LIN {X 0,Y 624.18,Z 1233.226,A -85,B 0,C 180,E1 28878.176,E2 28878.176} C_VEL
LIN {X 0,Y 624.369,Z 1226.316,A -85,B 0,C 180,E1 28876.192,E2 28876.192} C_VEL
LIN {X 0,Y 624.711,Z 1218.668,A -85,B 0,C 180,E1 28874.303,E2 28874.303} C_VEL
LIN {X 0,Y 625.236,Z 1208.486,A -85,B 0,C 180,E1 28872.115,E2 28872.115} C_VEL
LIN {X 0,Y 626.088,Z 1194.972,A -85,B 0,C 180,E1 28869.622,E2 28869.622} C_VEL
LIN {X 0,Y 627.007,Z 1182.374,A -85,B 0,C 180,E1 28867.593,E2 28867.593} C_VEL
LIN {X 0,Y 628.175,Z 1168.153,A -85,B 0,C 180,E1 28865.55,E2 28865.55} C_VEL
LIN {X 0,Y 629.836,Z 1149.568,A -85,B 0,C 180,E1 28863.198,E2 28863.198} C_VEL
LIN {X 0,Y 631.397,Z 1133.289,A -85,B 0,C 180,E1 28861.374,E2 28861.374} C_VEL
LIN {X 0,Y 633.134,Z 1116.14,A -85,B 0,C 180,E1 28859.642,E2 28859.642} C_VEL
LIN {X 0,Y 635.523,Z 1093.346,A -85,B 0,C 180,E1 28857.604,E2 28857.604} C_VEL
LIN {X 0,Y 637.441,Z 1075.082,A -85,B 0,C 180,E1 28856.159,E2 28856.159} C_VEL
LIN {X 0,Y 639.341,Z 1056.883,A -85,B 0,C 180,E1 28854.861,E2 28854.861} C_VEL
LIN {X 0,Y 641.452,Z 1036.313,A -85,B 0,C 180,E1 28853.547,E2 28853.547} C_VEL
LIN {X 0,Y 643.934,Z 1010.451,A -85,B 0,C 180,E1 28852.109,E2 28852.109} C_VEL
LIN {X 0,Y 645.904,Z 988.416,A -85,B 0,C 180,E1 28851.057,E2 28851.057} C_VEL
LIN {X 0,Y 647.711,Z 966.655,A -85,B 0,C 180,E1 28850.157,E2 28850.157} C_VEL
LIN {X 0,Y 649.668,Z 941.07,A -85,B 0,C 180,E1 28849.262,E2 28849.262} C_VEL
LIN {X 0,Y 651.274,Z 914.57,A -85,B 0,C 180,E1 28848.527,E2 28848.527} C_VEL
LIN {X 0,Y 652.424,Z 891.793,A -85,B 0,C 180,E1 28848.029,E2 28848.029} C_VEL
LIN {X 0,Y 653.308,Z 868.616,A -85,B 0,C 180,E1 28847.646,E2 28847.646} C_VEL
LIN {X 0,Y 657.558,Z 645.724,A -85,B 0,C 180,E1 28844.671,E2 28844.671} C_VEL
LIN {X 0,Y 661.46,Z 453.662,A -85,B 0,C 180,E1 28842.041,E2 28842.041} C_VEL
LIN {X 0,Y 652.442,Z 440.492,A -85,B 0,C 180,E1 28840.932,E2 28840.932} C_VEL
LIN {X 0,Y 640.565,Z 424.796,A -85,B 0,C 180,E1 28839.411,E2 28839.411} C_VEL
LIN {X 0,Y 636.522,Z 419.568,A -85,B 0,C 180,E1 28838.871,E2 28838.871} C_VEL
LIN {X 0,Y 632.798,Z 414.661,A -85,B 0,C 180,E1 28838.359,E2 28838.359} C_VEL
LIN {X 0,Y 629.914,Z 411.091,A -85,B 0,C 180,E1 28837.959,E2 28837.959} C_VEL
LIN {X 0,Y 628.864,Z 409.317,A -85,B 0,C 180,E1 28837.803,E2 28837.803} C_VEL
LIN {X 0,Y 626.22,Z 406.822,A -85,B 0,C 180,E1 28837.441,E2 28837.441} C_VEL
LIN {X 0,Y 624.999,Z 403.732,A -85,B 0,C 180,E1 28837.236,E2 28837.236} C_VEL
LIN {X 0,Y 624.947,Z 403.381,A -85,B 0,C 180,E1 28837.174,E2 28837.174} C_VEL
LIN {X 0,Y 624.942,Z 403.357,A -85,B 0,C 180,E1 28833.945,E2 28833.945} C_VEL
LIN {X 0,Y 624.938,Z 403.354,A -85,B 0,C 180,E1 28830.772,E2 28830.772} C_VEL
LIN {X 0,Y 624.939,Z 403.385,A -85,B 0,C 180,E1 28827.645,E2 28827.645} C_VEL
LIN {X 0,Y 624.94,Z 403.362,A -85,B 0,C 180,E1 28824.481,E2 28824.481} C_VEL
LIN {X 0,Y 624.932,Z 403.364,A -85,B 0,C 180,E1 28821.375,E2 28821.375} C_VEL
LIN {X 0,Y 624.944,Z 403.382,A -85,B 0,C 180,E1 28818.276,E2 28818.276} C_VEL
LIN {X 0,Y 624.926,Z 403.352,A -85,B 0,C 180,E1 28815.118,E2 28815.118} C_VEL
LIN {X 0,Y 624.945,Z 403.387,A -85,B 0,C 180,E1 28812.005,E2 28812.005} C_VEL
LIN {X 0,Y 624.923,Z 403.347,A -85,B 0,C 180,E1 28808.836,E2 28808.836} C_VEL
LIN {X 0,Y 624.946,Z 403.385,A -85,B 0,C 180,E1 28805.785,E2 28805.785} C_VEL
LIN {X 0,Y 624.921,Z 403.345,A -85,B 0,C 180,E1 28802.66,E2 28802.66} C_VEL
LIN {X 0,Y 624.949,Z 403.386,A -85,B 0,C 180,E1 28799.633,E2 28799.633} C_VEL
LIN {X 0,Y 624.922,Z 403.343,A -85,B 0,C 180,E1 28796.514,E2 28796.514} C_VEL
LIN {X 0,Y 624.948,Z 403.382,A -85,B 0,C 180,E1 28793.385,E2 28793.385} C_VEL
LIN {X 0,Y 624.918,Z 403.35,A -85,B 0,C 180,E1 28790.235,E2 28790.235} C_VEL
LIN {X 0,Y 624.949,Z 403.377,A -85,B 0,C 180,E1 28787.15,E2 28787.15} C_VEL
LIN {X 0,Y 624.919,Z 403.366,A -85,B 0,C 180,E1 28784.026,E2 28784.026} C_VEL
LIN {X 0,Y 624.948,Z 403.363,A -85,B 0,C 180,E1 28780.95,E2 28780.95} C_VEL
LIN {X 0,Y 624.918,Z 403.383,A -85,B 0,C 180,E1 28777.814,E2 28777.814} C_VEL
LIN {X 0,Y 624.947,Z 403.352,A -85,B 0,C 180,E1 28774.711,E2 28774.711} C_VEL
LIN {X 0,Y 624.917,Z 403.38,A -85,B 0,C 180,E1 28771.627,E2 28771.627} C_VEL
LIN {X 0,Y 624.954,Z 403.379,A -85,B 0,C 180,E1 28768.561,E2 28768.561} C_VEL
LIN {X 0,Y 624.916,Z 403.363,A -85,B 0,C 180,E1 28765.388,E2 28765.388} C_VEL
LIN {X 0,Y 624.957,Z 403.626,A -85,B 0,C 180,E1 28764.832,E2 28764.832} C_VEL
LIN {X 0,Y 626.263,Z 406.877,A -85,B 0,C 180,E1 28764.355,E2 28764.355} C_VEL
LIN {X 0,Y 627.353,Z 408.515,A -85,B 0,C 180,E1 28764.065,E2 28764.065} C_VEL
LIN {X 0,Y 629.05,Z 412.084,A -85,B 0,C 180,E1 28763.524,E2 28763.524} C_VEL
LIN {X 0,Y 634.263,Z 422.738,A -85,B 0,C 180,E1 28761.946,E2 28761.946} C_VEL
LIN {X 0,Y 636.116,Z 426.172,A -85,B 0,C 180,E1 28761.475,E2 28761.475} C_VEL
LIN {X 0,Y 652.475,Z 449.581,A -85,B 0,C 180,E1 28759.332,E2 28759.332} C_VEL
LIN {X 0,Y 661.483,Z 463.146,A -85,B 0,C 180,E1 28758.223,E2 28758.223} C_VEL
LIN {X 0,Y 661.775,Z 465.886,A -85,B 0,C 180,E1 28758.151,E2 28758.151} C_VEL
LIN {X 0,Y 657.599,Z 673.657,A -85,B 0,C 180,E1 28755.311,E2 28755.311} C_VEL
LIN {X 0,Y 653.346,Z 897.515,A -85,B 0,C 180,E1 28752.325,E2 28752.325} C_VEL
LIN {X 0,Y 652.452,Z 921.239,A -85,B 0,C 180,E1 28751.936,E2 28751.936} C_VEL
LIN {X 0,Y 651.313,Z 943.825,A -85,B 0,C 180,E1 28751.446,E2 28751.446} C_VEL
LIN {X 0,Y 649.785,Z 969.298,A -85,B 0,C 180,E1 28750.747,E2 28750.747} C_VEL
LIN {X 0,Y 647.795,Z 995.651,A -85,B 0,C 180,E1 28749.836,E2 28749.836} C_VEL
LIN {X 0,Y 645.982,Z 1017.523,A -85,B 0,C 180,E1 28748.937,E2 28748.937} C_VEL
LIN {X 0,Y 644.092,Z 1038.646,A -85,B 0,C 180,E1 28747.936,E2 28747.936} C_VEL
LIN {X 0,Y 641.751,Z 1063.464,A -85,B 0,C 180,E1 28746.584,E2 28746.584} C_VEL
LIN {X 0,Y 639.401,Z 1086.279,A -85,B 0,C 180,E1 28745.136,E2 28745.136} C_VEL
LIN {X 0,Y 637.5,Z 1104.526,A -85,B 0,C 180,E1 28743.838,E2 28743.838} C_VEL
LIN {X 0,Y 635.638,Z 1122.229,A -85,B 0,C 180,E1 28742.442,E2 28742.442} C_VEL
LIN {X 0,Y 633.467,Z 1143.165,A -85,B 0,C 180,E1 28740.603,E2 28740.603} C_VEL
LIN {X 0,Y 631.479,Z 1162.423,A -85,B 0,C 180,E1 28738.673,E2 28738.673} C_VEL
LIN {X 0,Y 629.929,Z 1178.632,A -85,B 0,C 180,E1 28736.865,E2 28736.865} C_VEL
LIN {X 0,Y 628.322,Z 1196.412,A -85,B 0,C 180,E1 28734.644,E2 28734.644} C_VEL
LIN {X 0,Y 627.081,Z 1211.45,A -85,B 0,C 180,E1 28732.503,E2 28732.503} C_VEL
LIN {X 0,Y 626.139,Z 1224.134,A -85,B 0,C 180,E1 28730.474,E2 28730.474} C_VEL
LIN {X 0,Y 625.299,Z 1237.338,A -85,B 0,C 180,E1 28728.076,E2 28728.076} C_VEL
LIN {X 0,Y 624.747,Z 1248.064,A -85,B 0,C 180,E1 28725.791,E2 28725.791} C_VEL
LIN {X 0,Y 624.373,Z 1256.146,A -85,B 0,C 180,E1 28723.808,E2 28723.808} C_VEL
LIN {X 0,Y 624.185,Z 1262.738,A -85,B 0,C 180,E1 28721.929,E2 28721.929} C_VEL
LIN {X 0,Y 624.025,Z 1268.81,A -85,B 0,C 180,E1 28719.876,E2 28719.876} C_VEL
LIN {X 0,Y 623.936,Z 1274.143,A -85,B 0,C 180,E1 28717.647,E2 28717.647} C_VEL
LIN {X 0,Y 623.92,Z 1278.422,A -85,B 0,C 180,E1 28715.153,E2 28715.153} C_VEL
LIN {X 0,Y 623.91,Z 1280.741,A -85,B 0,C 180,E1 28712.944,E2 28712.944} C_VEL
LIN {X 0,Y 623.875,Z 1281.759,A -85,B 0,C 180,E1 28711.014,E2 28711.014} C_VEL
LIN {X 0,Y 623.865,Z 1281.806,A -85,B 0,C 180,E1 28709.178,E2 28709.178} C_VEL
LIN {X 0,Y 623.909,Z 1280.95,A -85,B 0,C 180,E1 28707.341,E2 28707.341} C_VEL
LIN {X 0,Y 623.915,Z 1278.904,A -85,B 0,C 180,E1 28705.224,E2 28705.224} C_VEL
LIN {X 0,Y 623.953,Z 1275.087,A -85,B 0,C 180,E1 28702.824,E2 28702.824} C_VEL
LIN {X 0,Y 623.985,Z 1269.85,A -85,B 0,C 180,E1 28700.505,E2 28700.505} C_VEL
LIN {X 0,Y 624.178,Z 1263.371,A -85,B 0,C 180,E1 28698.266,E2 28698.266} C_VEL
LIN {X 0,Y 624.361,Z 1256.533,A -85,B 0,C 180,E1 28696.295,E2 28696.295} C_VEL
LIN {X 0,Y 624.7,Z 1248.923,A -85,B 0,C 180,E1 28694.407,E2 28694.407} C_VEL
LIN {X 0,Y 625.201,Z 1239.245,A -85,B 0,C 180,E1 28692.315,E2 28692.315} C_VEL
LIN {X 0,Y 626.033,Z 1225.91,A -85,B 0,C 180,E1 28689.824,E2 28689.824} C_VEL
LIN {X 0,Y 627.001,Z 1212.516,A -85,B 0,C 180,E1 28687.66,E2 28687.66} C_VEL
LIN {X 0,Y 628.135,Z 1198.609,A -85,B 0,C 180,E1 28685.658,E2 28685.658} C_VEL
LIN {X 0,Y 629.782,Z 1180.116,A -85,B 0,C 180,E1 28683.307,E2 28683.307} C_VEL
LIN {X 0,Y 631.386,Z 1163.434,A -85,B 0,C 180,E1 28681.435,E2 28681.435} C_VEL
LIN {X 0,Y 633.123,Z 1146.245,A -85,B 0,C 180,E1 28679.697,E2 28679.697} C_VEL
LIN {X 0,Y 635.505,Z 1123.499,A -85,B 0,C 180,E1 28677.662,E2 28677.662} C_VEL
LIN {X 0,Y 637.379,Z 1105.658,A -85,B 0,C 180,E1 28676.247,E2 28676.247} C_VEL
LIN {X 0,Y 639.312,Z 1087.141,A -85,B 0,C 180,E1 28674.924,E2 28674.924} C_VEL
LIN {X 0,Y 641.394,Z 1066.854,A -85,B 0,C 180,E1 28673.625,E2 28673.625} C_VEL
LIN {X 0,Y 643.903,Z 1040.838,A -85,B 0,C 180,E1 28672.174,E2 28672.174} C_VEL
LIN {X 0,Y 645.857,Z 1018.977,A -85,B 0,C 180,E1 28671.127,E2 28671.127} C_VEL
LIN {X 0,Y 647.601,Z 998.036,A -85,B 0,C 180,E1 28670.256,E2 28670.256} C_VEL
LIN {X 0,Y 649.259,Z 976.12,A -85,B 0,C 180,E1 28669.474,E2 28669.474} C_VEL
LIN {X 0,Y 651.057,Z 948.853,A -85,B 0,C 180,E1 28668.675,E2 28668.675} C_VEL
LIN {X 0,Y 652.353,Z 923.503,A -85,B 0,C 180,E1 28668.107,E2 28668.107} C_VEL
LIN {X 0,Y 653.236,Z 900.82,A -85,B 0,C 180,E1 28667.723,E2 28667.723} C_VEL
LIN {X 0,Y 657.425,Z 682.671,A -85,B 0,C 180,E1 28664.81,E2 28664.81} C_VEL
LIN {X 0,Y 661.622,Z 473.319,A -85,B 0,C 180,E1 28661.952,E2 28661.952} C_VEL
LIN {X 0,Y 661.642,Z 463.826,A -85,B 0,C 180,E1 28661.803,E2 28661.803} C_VEL
LIN {X 0,Y 660.917,Z 462.029,A -85,B 0,C 180,E1 28661.705,E2 28661.705} C_VEL
LIN {X 0,Y 647.235,Z 442.165,A -85,B 0,C 180,E1 28660.005,E2 28660.005} C_VEL
LIN {X 0,Y 635.569,Z 425.222,A -85,B 0,C 180,E1 28658.42,E2 28658.42} C_VEL
LIN {X 0,Y 630.828,Z 415.845,A -85,B 0,C 180,E1 28657.036,E2 28657.036} C_VEL
LIN {X 0,Y 628.688,Z 411.575,A -85,B 0,C 180,E1 28656.387,E2 28656.387} C_VEL
LIN {X 0,Y 626.981,Z 407.792,A -85,B 0,C 180,E1 28655.823,E2 28655.823} C_VEL
LIN {X 0,Y 625.107,Z 404.452,A -85,B 0,C 180,E1 28655.271,E2 28655.271} C_VEL
LIN {X 0,Y 624.89,Z 403.378,A -85,B 0,C 180,E1 28655.101,E2 28655.101} C_VEL
LIN {X 0,Y 624.932,Z 403.383,A -85,B 0,C 180,E1 28652.191,E2 28652.191} C_VEL
LIN {X 0,Y 624.885,Z 403.365,A -85,B 0,C 180,E1 28649.107,E2 28649.107} C_VEL
LIN {X 0,Y 624.886,Z 403.376,A -85,B 0,C 180,E1 28646.413,E2 28646.413} C_VEL
LIN {X 0,Y 624.898,Z 403.391,A -85,B 0,C 180,E1 28643.18,E2 28643.18} C_VEL
LIN {X 0,Y 624.865,Z 403.359,A -85,B 0,C 180,E1 28640.514,E2 28640.514} C_VEL
LIN {X 0,Y 624.944,Z 403.389,A -85,B 0,C 180,E1 28637.505,E2 28637.505} C_VEL
LIN {X 0,Y 624.855,Z 403.36,A -85,B 0,C 180,E1 28634.537,E2 28634.537} C_VEL
LIN {X 0,Y 624.882,Z 403.392,A -85,B 0,C 180,E1 28631.819,E2 28631.819} C_VEL
LIN {X 0,Y 624.852,Z 403.363,A -85,B 0,C 180,E1 28628.586,E2 28628.586} C_VEL
LIN {X 0,Y 624.848,Z 403.394,A -85,B 0,C 180,E1 28626.063,E2 28626.063} C_VEL
LIN {X 0,Y 624.921,Z 403.351,A -85,B 0,C 180,E1 28623.027,E2 28623.027} C_VEL
LIN {X 0,Y 624.858,Z 403.393,A -85,B 0,C 180,E1 28620.092,E2 28620.092} C_VEL
LIN {X 0,Y 624.91,Z 403.353,A -85,B 0,C 180,E1 28617.249,E2 28617.249} C_VEL
LIN {X 0,Y 624.872,Z 403.391,A -85,B 0,C 180,E1 28614.122,E2 28614.122} C_VEL
LIN {X 0,Y 624.883,Z 403.359,A -85,B 0,C 180,E1 28611.442,E2 28611.442} C_VEL
LIN {X 0,Y 624.896,Z 403.389,A -85,B 0,C 180,E1 28608.181,E2 28608.181} C_VEL
LIN {X 0,Y 624.883,Z 403.358,A -85,B 0,C 180,E1 28605.45,E2 28605.45} C_VEL
LIN {X 0,Y 624.936,Z 403.386,A -85,B 0,C 180,E1 28602.302,E2 28602.302} C_VEL
LIN {X 0,Y 624.888,Z 403.354,A -85,B 0,C 180,E1 28599.38,E2 28599.38} C_VEL
LIN {X 0,Y 624.954,Z 403.378,A -85,B 0,C 180,E1 28596.323,E2 28596.323} C_VEL
LIN {X 0,Y 624.898,Z 403.371,A -85,B 0,C 180,E1 28593.28,E2 28593.28} C_VEL
LIN {X 0,Y 624.953,Z 403.353,A -85,B 0,C 180,E1 28590.265,E2 28590.265} C_VEL
LIN {X 0,Y 624.908,Z 403.391,A -85,B 0,C 180,E1 28587.151,E2 28587.151} C_VEL
LIN {X 0,Y 624.951,Z 403.371,A -85,B 0,C 180,E1 28584.042,E2 28584.042} C_VEL
LIN {X 0,Y 624.961,Z 403.612,A -85,B 0,C 180,E1 28582.679,E2 28582.679} C_VEL
LIN {X 0,Y 626.132,Z 406.672,A -85,B 0,C 180,E1 28582.48,E2 28582.48} C_VEL
LIN {X 0,Y 628.699,Z 409.185,A -85,B 0,C 180,E1 28582.128,E2 28582.128} C_VEL
LIN {X 0,Y 629.507,Z 410.299,A -85,B 0,C 180,E1 28582.012,E2 28582.012} C_VEL
LIN {X 0,Y 632.071,Z 413.977,A -85,B 0,C 180,E1 28581.646,E2 28581.646} C_VEL
LIN {X 0,Y 633.818,Z 415.911,A -85,B 0,C 180,E1 28581.411,E2 28581.411} C_VEL
LIN {X 0,Y 637.218,Z 420.26,A -85,B 0,C 180,E1 28580.949,E2 28580.949} C_VEL
LIN {X 0,Y 651.261,Z 439.003,A -85,B 0,C 180,E1 28579.123,E2 28579.123} C_VEL
LIN {X 0,Y 660.214,Z 451.648,A -85,B 0,C 180,E1 28578.022,E2 28578.022} C_VEL
LIN {X 0,Y 661.481,Z 454.083,A -85,B 0,C 180,E1 28577.86,E2 28577.86} C_VEL
LIN {X 0,Y 660.474,Z 501.439,A -85,B 0,C 180,E1 28577.206,E2 28577.206} C_VEL
LIN {X 0,Y 659.621,Z 509.147,A -85,B 0,C 180,E1 28577.165,E2 28577.165} C_VEL
LIN {X 0,Y 654.944,Z 529.83,A -85,B 0,C 180,E1 28577.283,E2 28577.283} C_VEL
LIN {X 0,Y 654.301,Z 536.437,A -85,B 0,C 180,E1 28577.239,E2 28577.239} C_VEL
LIN {X 0,Y 649.641,Z 757.843,A -85,B 0,C 180,E1 28574.227,E2 28574.227} C_VEL
LIN {X 0,Y 647.176,Z 874.928,A -85,B 0,C 180,E1 28572.649,E2 28572.649} C_VEL
LIN {X 0,Y 646,Z 902.071,A -85,B 0,C 180,E1 28572.153,E2 28572.153} C_VEL
LIN {X 0,Y 644.375,Z 928.231,A -85,B 0,C 180,E1 28571.496,E2 28571.496} C_VEL
LIN {X 0,Y 642.849,Z 949.425,A -85,B 0,C 180,E1 28570.839,E2 28570.839} C_VEL
LIN {X 0,Y 641.18,Z 970.031,A -85,B 0,C 180,E1 28570.087,E2 28570.087} C_VEL
LIN {X 0,Y 639.218,Z 992.171,A -85,B 0,C 180,E1 28569.145,E2 28569.145} C_VEL
LIN {X 0,Y 636.642,Z 1018.743,A -85,B 0,C 180,E1 28567.814,E2 28567.814} C_VEL
LIN {X 0,Y 634.448,Z 1039.446,A -85,B 0,C 180,E1 28566.613,E2 28566.613} C_VEL
LIN {X 0,Y 632.414,Z 1058.012,A -85,B 0,C 180,E1 28565.405,E2 28565.405} C_VEL
LIN {X 0,Y 630.33,Z 1076.763,A -85,B 0,C 180,E1 28564.046,E2 28564.046} C_VEL
LIN {X 0,Y 627.864,Z 1098.737,A -85,B 0,C 180,E1 28562.26,E2 28562.26} C_VEL
LIN {X 0,Y 625.641,Z 1118.412,A -85,B 0,C 180,E1 28560.432,E2 28560.432} C_VEL
LIN {X 0,Y 623.881,Z 1134.672,A -85,B 0,C 180,E1 28558.756,E2 28558.756} C_VEL
LIN {X 0,Y 621.996,Z 1153.107,A -85,B 0,C 180,E1 28556.641,E2 28556.641} C_VEL
LIN {X 0,Y 620.362,Z 1170.144,A -85,B 0,C 180,E1 28554.403,E2 28554.403} C_VEL
LIN {X 0,Y 619.177,Z 1183.762,A -85,B 0,C 180,E1 28552.396,E2 28552.396} C_VEL
LIN {X 0,Y 618.058,Z 1198.42,A -85,B 0,C 180,E1 28549.954,E2 28549.954} C_VEL
LIN {X 0,Y 617.254,Z 1210.428,A -85,B 0,C 180,E1 28547.628,E2 28547.628} C_VEL
LIN {X 0,Y 616.73,Z 1219.949,A -85,B 0,C 180,E1 28545.511,E2 28545.511} C_VEL
LIN {X 0,Y 616.358,Z 1228.838,A -85,B 0,C 180,E1 28543.218,E2 28543.218} C_VEL
LIN {X 0,Y 616.104,Z 1236.923,A -85,B 0,C 180,E1 28540.657,E2 28540.657} C_VEL
LIN {X 0,Y 615.995,Z 1242.642,A -85,B 0,C 180,E1 28538.396,E2 28538.396} C_VEL
LIN {X 0,Y 615.936,Z 1247.124,A -85,B 0,C 180,E1 28536.052,E2 28536.052} C_VEL
LIN {X 0,Y 615.913,Z 1250.306,A -85,B 0,C 180,E1 28533.532,E2 28533.532} C_VEL
LIN {X 0,Y 615.894,Z 1251.704,A -85,B 0,C 180,E1 28531.205,E2 28531.205} C_VEL
LIN {X 0,Y 615.864,Z 1251.837,A -85,B 0,C 180,E1 28529.252,E2 28529.252} C_VEL
LIN {X 0,Y 615.907,Z 1250.977,A -85,B 0,C 180,E1 28527.297,E2 28527.297} C_VEL
LIN {X 0,Y 615.915,Z 1248.946,A -85,B 0,C 180,E1 28525.153,E2 28525.153} C_VEL
LIN {X 0,Y 615.954,Z 1245.154,A -85,B 0,C 180,E1 28522.722,E2 28522.722} C_VEL
LIN {X 0,Y 616.007,Z 1239.693,A -85,B 0,C 180,E1 28520.278,E2 28520.278} C_VEL
LIN {X 0,Y 616.197,Z 1233.451,A -85,B 0,C 180,E1 28518.092,E2 28518.092} C_VEL
LIN {X 0,Y 616.402,Z 1226.667,A -85,B 0,C 180,E1 28516.105,E2 28516.105} C_VEL
LIN {X 0,Y 616.772,Z 1219.075,A -85,B 0,C 180,E1 28514.192,E2 28514.192} C_VEL
LIN {X 0,Y 617.303,Z 1209.416,A -85,B 0,C 180,E1 28512.073,E2 28512.073} C_VEL
LIN {X 0,Y 618.211,Z 1196.113,A -85,B 0,C 180,E1 28509.549,E2 28509.549} C_VEL
LIN {X 0,Y 619.232,Z 1183.003,A -85,B 0,C 180,E1 28507.396,E2 28507.396} C_VEL
LIN {X 0,Y 620.417,Z 1169.572,A -85,B 0,C 180,E1 28505.427,E2 28505.427} C_VEL
LIN {X 0,Y 622.116,Z 1151.935,A -85,B 0,C 180,E1 28503.129,E2 28503.129} C_VEL
LIN {X 0,Y 623.88,Z 1134.67,A -85,B 0,C 180,E1 28501.154,E2 28501.154} C_VEL
LIN {X 0,Y 625.64,Z 1118.409,A -85,B 0,C 180,E1 28499.477,E2 28499.477} C_VEL
LIN {X 0,Y 627.941,Z 1098.152,A -85,B 0,C 180,E1 28497.598,E2 28497.598} C_VEL
LIN {X 0,Y 630.37,Z 1076.407,A -85,B 0,C 180,E1 28495.837,E2 28495.837} C_VEL
LIN {X 0,Y 632.454,Z 1057.679,A -85,B 0,C 180,E1 28494.482,E2 28494.482} C_VEL
LIN {X 0,Y 634.5,Z 1038.978,A -85,B 0,C 180,E1 28493.268,E2 28493.268} C_VEL
LIN {X 0,Y 637.003,Z 1015.386,A -85,B 0,C 180,E1 28491.909,E2 28491.909} C_VEL
LIN {X 0,Y 639.342,Z 990.659,A -85,B 0,C 180,E1 28490.697,E2 28490.697} C_VEL
LIN {X 0,Y 641.244,Z 969.205,A -85,B 0,C 180,E1 28489.791,E2 28489.791} C_VEL
LIN {X 0,Y 642.921,Z 948.454,A -85,B 0,C 180,E1 28489.038,E2 28489.038} C_VEL
LIN {X 0,Y 644.672,Z 924.03,A -85,B 0,C 180,E1 28488.293,E2 28488.293} C_VEL
LIN {X 0,Y 646.263,Z 895.924,A -85,B 0,C 180,E1 28487.633,E2 28487.633} C_VEL
LIN {X 0,Y 647.247,Z 872.707,A -85,B 0,C 180,E1 28487.228,E2 28487.228} C_VEL
LIN {X 0,Y 651.601,Z 661.791,A -85,B 0,C 180,E1 28484.388,E2 28484.388} C_VEL
LIN {X 0,Y 656.051,Z 457.437,A -85,B 0,C 180,E1 28481.572,E2 28481.572} C_VEL
LIN {X 0,Y 645.173,Z 442.024,A -85,B 0,C 180,E1 28480.203,E2 28480.203} C_VEL
LIN {X 0,Y 633.088,Z 426.146,A -85,B 0,C 180,E1 28478.599,E2 28478.599} C_VEL
LIN {X 0,Y 629.106,Z 421.023,A -85,B 0,C 180,E1 28478.045,E2 28478.045} C_VEL
LIN {X 0,Y 625.872,Z 416.621,A -85,B 0,C 180,E1 28477.581,E2 28477.581} C_VEL
LIN {X 0,Y 622.34,Z 412.611,A -85,B 0,C 180,E1 28477.078,E2 28477.078} C_VEL
LIN {X 0,Y 621.204,Z 410.46,A -85,B 0,C 180,E1 28476.897,E2 28476.897} C_VEL
LIN {X 0,Y 618.464,Z 408.085,A -85,B 0,C 180,E1 28476.51,E2 28476.51} C_VEL
LIN {X 0,Y 617.116,Z 405.016,A -85,B 0,C 180,E1 28476.28,E2 28476.28} C_VEL
LIN {X 0,Y 617.01,Z 404.371,A -85,B 0,C 180,E1 28476.227,E2 28476.227} C_VEL
LIN {X 0,Y 617.009,Z 404.366,A -85,B 0,C 180,E1 28472.991,E2 28472.991} C_VEL
LIN {X 0,Y 616.998,Z 404.342,A -85,B 0,C 180,E1 28469.729,E2 28469.729} C_VEL
LIN {X 0,Y 617.004,Z 404.351,A -85,B 0,C 180,E1 28466.673,E2 28466.673} C_VEL
LIN {X 0,Y 616.996,Z 404.37,A -85,B 0,C 180,E1 28463.47,E2 28463.47} C_VEL
LIN {X 0,Y 617.004,Z 404.337,A -85,B 0,C 180,E1 28460.391,E2 28460.391} C_VEL
LIN {X 0,Y 616.995,Z 404.373,A -85,B 0,C 180,E1 28457.252,E2 28457.252} C_VEL
LIN {X 0,Y 617.005,Z 404.339,A -85,B 0,C 180,E1 28454.164,E2 28454.164} C_VEL
LIN {X 0,Y 616.993,Z 404.372,A -85,B 0,C 180,E1 28451.025,E2 28451.025} C_VEL
LIN {X 0,Y 617.002,Z 404.343,A -85,B 0,C 180,E1 28447.824,E2 28447.824} C_VEL
LIN {X 0,Y 616.986,Z 404.369,A -85,B 0,C 180,E1 28444.666,E2 28444.666} C_VEL
LIN {X 0,Y 617.003,Z 404.348,A -85,B 0,C 180,E1 28441.486,E2 28441.486} C_VEL
LIN {X 0,Y 616.983,Z 404.365,A -85,B 0,C 180,E1 28438.421,E2 28438.421} C_VEL
LIN {X 0,Y 617.003,Z 404.35,A -85,B 0,C 180,E1 28435.259,E2 28435.259} C_VEL
LIN {X 0,Y 616.98,Z 404.359,A -85,B 0,C 180,E1 28432.176,E2 28432.176} C_VEL
LIN {X 0,Y 617.007,Z 404.357,A -85,B 0,C 180,E1 28429.07,E2 28429.07} C_VEL
LIN {X 0,Y 616.977,Z 404.349,A -85,B 0,C 180,E1 28425.931,E2 28425.931} C_VEL
LIN {X 0,Y 617.01,Z 404.373,A -85,B 0,C 180,E1 28422.846,E2 28422.846} C_VEL
LIN {X 0,Y 616.975,Z 404.34,A -85,B 0,C 180,E1 28419.707,E2 28419.707} C_VEL
LIN {X 0,Y 617.01,Z 404.367,A -85,B 0,C 180,E1 28416.607,E2 28416.607} C_VEL
LIN {X 0,Y 616.975,Z 404.363,A -85,B 0,C 180,E1 28413.43,E2 28413.43} C_VEL
LIN {X 0,Y 617.01,Z 404.339,A -85,B 0,C 180,E1 28410.379,E2 28410.379} C_VEL
LIN {X 0,Y 616.972,Z 404.36,A -85,B 0,C 180,E1 28407.26,E2 28407.26} C_VEL
LIN {X 0,Y 617.022,Z 404.501,A -85,B 0,C 180,E1 28405.758,E2 28405.758} C_VEL
LIN {X 0,Y 618.161,Z 407.659,A -85,B 0,C 180,E1 28405.294,E2 28405.294} C_VEL
LIN {X 0,Y 619.485,Z 409.717,A -85,B 0,C 180,E1 28404.921,E2 28404.921} C_VEL
LIN {X 0,Y 626.365,Z 423.493,A -85,B 0,C 180,E1 28402.77,E2 28402.77} C_VEL
LIN {X 0,Y 627.636,Z 425.839,A -85,B 0,C 180,E1 28402.456,E2 28402.456} C_VEL
LIN {X 0,Y 639.368,Z 442.419,A -85,B 0,C 180,E1 28400.831,E2 28400.831} C_VEL
LIN {X 0,Y 652.071,Z 460.969,A -85,B 0,C 180,E1 28399.185,E2 28399.185} C_VEL
LIN {X 0,Y 656.372,Z 467.664,A -85,B 0,C 180,E1 28398.648,E2 28398.648} C_VEL
LIN {X 0,Y 651.927,Z 675.488,A -85,B 0,C 180,E1 28395.788,E2 28395.788} C_VEL
LIN {X 0,Y 647.408,Z 898.124,A -85,B 0,C 180,E1 28392.795,E2 28392.795} C_VEL
LIN {X 0,Y 646.478,Z 921.376,A -85,B 0,C 180,E1 28392.41,E2 28392.41} C_VEL
LIN {X 0,Y 645.285,Z 943.689,A -85,B 0,C 180,E1 28391.924,E2 28391.924} C_VEL
LIN {X 0,Y 643.695,Z 968.754,A -85,B 0,C 180,E1 28391.235,E2 28391.235} C_VEL
LIN {X 0,Y 641.555,Z 995.648,A -85,B 0,C 180,E1 28390.303,E2 28390.303} C_VEL
LIN {X 0,Y 639.631,Z 1017.52,A -85,B 0,C 180,E1 28389.398,E2 28389.398} C_VEL
LIN {X 0,Y 637.621,Z 1038.642,A -85,B 0,C 180,E1 28388.391,E2 28388.391} C_VEL
LIN {X 0,Y 635.13,Z 1063.241,A -85,B 0,C 180,E1 28387.044,E2 28387.044} C_VEL
LIN {X 0,Y 632.686,Z 1085.542,A -85,B 0,C 180,E1 28385.62,E2 28385.62} C_VEL
LIN {X 0,Y 630.632,Z 1103.964,A -85,B 0,C 180,E1 28384.303,E2 28384.303} C_VEL
LIN {X 0,Y 628.588,Z 1122.227,A -85,B 0,C 180,E1 28382.852,E2 28382.852} C_VEL
LIN {X 0,Y 626.236,Z 1143.381,A -85,B 0,C 180,E1 28380.973,E2 28380.973} C_VEL
LIN {X 0,Y 624.107,Z 1162.421,A -85,B 0,C 180,E1 28379.044,E2 28379.044} C_VEL
LIN {X 0,Y 622.479,Z 1178.347,A -85,B 0,C 180,E1 28377.248,E2 28377.248} C_VEL
LIN {X 0,Y 620.774,Z 1195.704,A -85,B 0,C 180,E1 28375.066,E2 28375.066} C_VEL
LIN {X 0,Y 619.363,Z 1211.448,A -85,B 0,C 180,E1 28372.799,E2 28372.799} C_VEL
LIN {X 0,Y 618.339,Z 1224.132,A -85,B 0,C 180,E1 28370.744,E2 28370.744} C_VEL
LIN {X 0,Y 617.427,Z 1237.339,A -85,B 0,C 180,E1 28368.314,E2 28368.314} C_VEL
LIN {X 0,Y 616.835,Z 1248.065,A -85,B 0,C 180,E1 28365.999,E2 28365.999} C_VEL
LIN {X 0,Y 616.422,Z 1256.147,A -85,B 0,C 180,E1 28363.99,E2 28363.99} C_VEL
LIN {X 0,Y 616.209,Z 1262.738,A -85,B 0,C 180,E1 28362.086,E2 28362.086} C_VEL
LIN {X 0,Y 616.049,Z 1268.809,A -85,B 0,C 180,E1 28360.005,E2 28360.005} C_VEL
LIN {X 0,Y 615.939,Z 1274.339,A -85,B 0,C 180,E1 28357.653,E2 28357.653} C_VEL
LIN {X 0,Y 615.92,Z 1278.547,A -85,B 0,C 180,E1 28355.127,E2 28355.127} C_VEL
LIN {X 0,Y 615.91,Z 1280.741,A -85,B 0,C 180,E1 28352.982,E2 28352.982} C_VEL
LIN {X 0,Y 615.876,Z 1281.758,A -85,B 0,C 180,E1 28351.027,E2 28351.027} C_VEL
LIN {X 0,Y 615.866,Z 1281.806,A -85,B 0,C 180,E1 28349.167,E2 28349.167} C_VEL
LIN {X 0,Y 615.909,Z 1280.95,A -85,B 0,C 180,E1 28347.306,E2 28347.306} C_VEL
LIN {X 0,Y 615.915,Z 1279.015,A -85,B 0,C 180,E1 28345.255,E2 28345.255} C_VEL
LIN {X 0,Y 615.953,Z 1275.43,A -85,B 0,C 180,E1 28342.918,E2 28342.918} C_VEL
LIN {X 0,Y 615.993,Z 1270.104,A -85,B 0,C 180,E1 28340.475,E2 28340.475} C_VEL
LIN {X 0,Y 616.193,Z 1263.674,A -85,B 0,C 180,E1 28338.207,E2 28338.207} C_VEL
LIN {X 0,Y 616.394,Z 1256.885,A -85,B 0,C 180,E1 28336.21,E2 28336.21} C_VEL
LIN {X 0,Y 616.759,Z 1249.329,A -85,B 0,C 180,E1 28334.297,E2 28334.297} C_VEL
LIN {X 0,Y 617.268,Z 1240.136,A -85,B 0,C 180,E1 28332.267,E2 28332.267} C_VEL
LIN {X 0,Y 618.116,Z 1227.612,A -85,B 0,C 180,E1 28329.851,E2 28329.851} C_VEL
LIN {X 0,Y 619.223,Z 1213.154,A -85,B 0,C 180,E1 28327.464,E2 28327.464} C_VEL
LIN {X 0,Y 620.441,Z 1199.321,A -85,B 0,C 180,E1 28325.437,E2 28325.437} C_VEL
LIN {X 0,Y 622.161,Z 1181.48,A -85,B 0,C 180,E1 28323.12,E2 28323.12} C_VEL
LIN {X 0,Y 623.913,Z 1164.358,A -85,B 0,C 180,E1 28321.165,E2 28321.165} C_VEL
LIN {X 0,Y 625.649,Z 1148.334,A -85,B 0,C 180,E1 28319.515,E2 28319.515} C_VEL
LIN {X 0,Y 627.987,Z 1127.778,A -85,B 0,C 180,E1 28317.61,E2 28317.61} C_VEL
LIN {X 0,Y 630.347,Z 1106.601,A -85,B 0,C 180,E1 28315.897,E2 28315.897} C_VEL
LIN {X 0,Y 632.431,Z 1087.872,A -85,B 0,C 180,E1 28314.54,E2 28314.54} C_VEL
LIN {X 0,Y 634.464,Z 1069.284,A -85,B 0,C 180,E1 28313.332,E2 28313.332} C_VEL
LIN {X 0,Y 636.771,Z 1047.548,A -85,B 0,C 180,E1 28312.074,E2 28312.074} C_VEL
LIN {X 0,Y 639.303,Z 1021.12,A -85,B 0,C 180,E1 28310.762,E2 28310.762} C_VEL
LIN {X 0,Y 641.202,Z 999.735,A -85,B 0,C 180,E1 28309.857,E2 28309.857} C_VEL
LIN {X 0,Y 642.875,Z 979.075,A -85,B 0,C 180,E1 28309.104,E2 28309.104} C_VEL
LIN {X 0,Y 644.529,Z 956.053,A -85,B 0,C 180,E1 28308.396,E2 28308.396} C_VEL
LIN {X 0,Y 646.194,Z 927.539,A -85,B 0,C 180,E1 28307.709,E2 28307.709} C_VEL
LIN {X 0,Y 647.227,Z 903.358,A -85,B 0,C 180,E1 28307.283,E2 28307.283} C_VEL
LIN {X 0,Y 651.521,Z 695.575,A -85,B 0,C 180,E1 28304.485,E2 28304.485} C_VEL
LIN {X 0,Y 656.055,Z 482.199,A -85,B 0,C 180,E1 28301.556,E2 28301.556} C_VEL
LIN {X 0,Y 656.281,Z 467.185,A -85,B 0,C 180,E1 28301.336,E2 28301.336} C_VEL
LIN {X 0,Y 640.84,Z 444.49,A -85,B 0,C 180,E1 28299.365,E2 28299.365} C_VEL
LIN {X 0,Y 630.462,Z 429.936,A -85,B 0,C 180,E1 28297.949,E2 28297.949} C_VEL
LIN {X 0,Y 626.958,Z 424.776,A -85,B 0,C 180,E1 28297.418,E2 28297.418} C_VEL
LIN {X 0,Y 621.219,Z 413.18,A -85,B 0,C 180,E1 28295.638,E2 28295.638} C_VEL
LIN {X 0,Y 619.341,Z 409.315,A -85,B 0,C 180,E1 28295.025,E2 28295.025} C_VEL
LIN {X 0,Y 617.316,Z 405.866,A -85,B 0,C 180,E1 28294.422,E2 28294.422} C_VEL
LIN {X 0,Y 616.997,Z 404.342,A -85,B 0,C 180,E1 28294.218,E2 28294.218} C_VEL
LIN {X 0,Y 616.951,Z 404.368,A -85,B 0,C 180,E1 28291.132,E2 28291.132} C_VEL
LIN {X 0,Y 616.961,Z 404.368,A -85,B 0,C 180,E1 28288.35,E2 28288.35} C_VEL
LIN {X 0,Y 616.945,Z 404.346,A -85,B 0,C 180,E1 28285.062,E2 28285.062} C_VEL
LIN {X 0,Y 616.945,Z 404.38,A -85,B 0,C 180,E1 28282.287,E2 28282.287} C_VEL
LIN {X 0,Y 616.945,Z 404.359,A -85,B 0,C 180,E1 28279.012,E2 28279.012} C_VEL
LIN {X 0,Y 616.924,Z 404.37,A -85,B 0,C 180,E1 28276.284,E2 28276.284} C_VEL
LIN {X 0,Y 616.979,Z 404.361,A -85,B 0,C 180,E1 28273.209,E2 28273.209} C_VEL
LIN {X 0,Y 616.908,Z 404.363,A -85,B 0,C 180,E1 28270.27,E2 28270.27} C_VEL
LIN {X 0,Y 617,Z 404.361,A -85,B 0,C 180,E1 28267.262,E2 28267.262} C_VEL
LIN {X 0,Y 616.908,Z 404.36,A -85,B 0,C 180,E1 28264.183,E2 28264.183} C_VEL
LIN {X 0,Y 617,Z 404.363,A -85,B 0,C 180,E1 28261.114,E2 28261.114} C_VEL
LIN {X 0,Y 616.921,Z 404.36,A -85,B 0,C 180,E1 28258.142,E2 28258.142} C_VEL
LIN {X 0,Y 616.97,Z 404.362,A -85,B 0,C 180,E1 28255.248,E2 28255.248} C_VEL
LIN {X 0,Y 616.939,Z 404.361,A -85,B 0,C 180,E1 28252.175,E2 28252.175} C_VEL
LIN {X 0,Y 616.952,Z 404.363,A -85,B 0,C 180,E1 28249.353,E2 28249.353} C_VEL
LIN {X 0,Y 616.953,Z 404.354,A -85,B 0,C 180,E1 28246.087,E2 28246.087} C_VEL
LIN {X 0,Y 616.957,Z 404.368,A -85,B 0,C 180,E1 28243.274,E2 28243.274} C_VEL
LIN {X 0,Y 616.97,Z 404.341,A -85,B 0,C 180,E1 28240.004,E2 28240.004} C_VEL
LIN {X 0,Y 616.967,Z 404.377,A -85,B 0,C 180,E1 28237.11,E2 28237.11} C_VEL
LIN {X 0,Y 616.978,Z 404.345,A -85,B 0,C 180,E1 28233.844,E2 28233.844} C_VEL
LIN {X 0,Y 616.978,Z 404.359,A -85,B 0,C 180,E1 28230.909,E2 28230.909} C_VEL
LIN {X 0,Y 616.981,Z 404.378,A -85,B 0,C 180,E1 28227.588,E2 28227.588} C_VEL
LIN {X 0,Y 616.999,Z 404.347,A -85,B 0,C 180,E1 28224.538,E2 28224.538} C_VEL
LIN {X 0,Y 617.026,Z 404.575,A -85,B 0,C 180,E1 28223.647,E2 28223.647} C_VEL
LIN {X 0,Y 618.175,Z 407.685,A -85,B 0,C 180,E1 28223.441,E2 28223.441} C_VEL
LIN {X 0,Y 620.75,Z 410.216,A -85,B 0,C 180,E1 28223.071,E2 28223.071} C_VEL
LIN {X 0,Y 621.618,Z 411.27,A -85,B 0,C 180,E1 28222.944,E2 28222.944} C_VEL
LIN {X 0,Y 624.19,Z 414.961,A -85,B 0,C 180,E1 28222.56,E2 28222.56} C_VEL
LIN {X 0,Y 626.043,Z 416.939,A -85,B 0,C 180,E1 28222.301,E2 28222.301} C_VEL
LIN {X 0,Y 629.367,Z 421.267,A -85,B 0,C 180,E1 28221.829,E2 28221.829} C_VEL
LIN {X 0,Y 639.06,Z 433.991,A -85,B 0,C 180,E1 28220.504,E2 28220.504} C_VEL
LIN {X 0,Y 650.027,Z 448.794,A -85,B 0,C 180,E1 28219.088,E2 28219.088} C_VEL
LIN {X 0,Y 656.061,Z 457.672,A -85,B 0,C 180,E1 28218.333,E2 28218.333} C_VEL
LIN {X 0,Y 654.301,Z 536.437,A -85,B 0,C 180,E1 28217.239,E2 28217.239} C_VEL
LIN {X 0,Y 653.465,Z 544.14,A -85,B 0,C 180,E1 28217.196,E2 28217.196} C_VEL
LIN {X 0,Y 648.743,Z 564.814,A -85,B 0,C 180,E1 28217.319,E2 28217.319} C_VEL
LIN {X 0,Y 648.07,Z 571.425,A -85,B 0,C 180,E1 28217.278,E2 28217.278} C_VEL
LIN {X 0,Y 643.309,Z 786.733,A -85,B 0,C 180,E1 28214.336,E2 28214.336} C_VEL
LIN {X 0,Y 641.278,Z 875.348,A -85,B 0,C 180,E1 28213.129,E2 28213.129} C_VEL
LIN {X 0,Y 640.003,Z 902.848,A -85,B 0,C 180,E1 28212.62,E2 28212.62} C_VEL
LIN {X 0,Y 638.311,Z 928.562,A -85,B 0,C 180,E1 28211.968,E2 28211.968} C_VEL
LIN {X 0,Y 636.724,Z 949.439,A -85,B 0,C 180,E1 28211.317,E2 28211.317} C_VEL
LIN {X 0,Y 634.955,Z 970.044,A -85,B 0,C 180,E1 28210.561,E2 28210.561} C_VEL
LIN {X 0,Y 632.845,Z 992.513,A -85,B 0,C 180,E1 28209.599,E2 28209.599} C_VEL
LIN {X 0,Y 630.149,Z 1018.645,A -85,B 0,C 180,E1 28208.281,E2 28208.281} C_VEL
LIN {X 0,Y 627.816,Z 1039.399,A -85,B 0,C 180,E1 28207.068,E2 28207.068} C_VEL
LIN {X 0,Y 625.643,Z 1058.018,A -85,B 0,C 180,E1 28205.847,E2 28205.847} C_VEL
LIN {X 0,Y 623.359,Z 1077.37,A -85,B 0,C 180,E1 28204.43,E2 28204.43} C_VEL
LIN {X 0,Y 620.617,Z 1100.109,A -85,B 0,C 180,E1 28202.548,E2 28202.548} C_VEL
LIN {X 0,Y 618.408,Z 1118.417,A -85,B 0,C 180,E1 28200.827,E2 28200.827} C_VEL
LIN {X 0,Y 616.543,Z 1134.427,A -85,B 0,C 180,E1 28199.159,E2 28199.159} C_VEL
LIN {X 0,Y 614.607,Z 1152.284,A -85,B 0,C 180,E1 28197.092,E2 28197.092} C_VEL
LIN {X 0,Y 612.78,Z 1169.72,A -85,B 0,C 180,E1 28194.788,E2 28194.788} C_VEL
LIN {X 0,Y 611.483,Z 1183.459,A -85,B 0,C 180,E1 28192.743,E2 28192.743} C_VEL
LIN {X 0,Y 610.283,Z 1197.902,A -85,B 0,C 180,E1 28190.319,E2 28190.319} C_VEL
LIN {X 0,Y 609.371,Z 1210.354,A -85,B 0,C 180,E1 28187.88,E2 28187.88} C_VEL
LIN {X 0,Y 608.818,Z 1219.786,A -85,B 0,C 180,E1 28185.757,E2 28185.757} C_VEL
LIN {X 0,Y 608.4,Z 1228.133,A -85,B 0,C 180,E1 28183.587,E2 28183.587} C_VEL
LIN {X 0,Y 608.128,Z 1236.413,A -85,B 0,C 180,E1 28180.99,E2 28180.99} C_VEL
LIN {X 0,Y 608.002,Z 1242.434,A -85,B 0,C 180,E1 28178.602,E2 28178.602} C_VEL
LIN {X 0,Y 607.942,Z 1246.963,A -85,B 0,C 180,E1 28176.227,E2 28176.227} C_VEL
LIN {X 0,Y 607.914,Z 1250.238,A -85,B 0,C 180,E1 28173.673,E2 28173.673} C_VEL
LIN {X 0,Y 607.895,Z 1251.704,A -85,B 0,C 180,E1 28171.221,E2 28171.221} C_VEL
LIN {X 0,Y 607.864,Z 1251.837,A -85,B 0,C 180,E1 28169.242,E2 28169.242} C_VEL
LIN {X 0,Y 607.908,Z 1250.977,A -85,B 0,C 180,E1 28167.262,E2 28167.262} C_VEL
LIN {X 0,Y 607.915,Z 1249.056,A -85,B 0,C 180,E1 28165.184,E2 28165.184} C_VEL
LIN {X 0,Y 607.956,Z 1245.497,A -85,B 0,C 180,E1 28162.816,E2 28162.816} C_VEL
LIN {X 0,Y 608.007,Z 1240.2,A -85,B 0,C 180,E1 28160.34,E2 28160.34} C_VEL
LIN {X 0,Y 608.218,Z 1233.485,A -85,B 0,C 180,E1 28157.945,E2 28157.945} C_VEL
LIN {X 0,Y 608.453,Z 1226.664,A -85,B 0,C 180,E1 28155.92,E2 28155.92} C_VEL
LIN {X 0,Y 608.89,Z 1218.632,A -85,B 0,C 180,E1 28153.876,E2 28153.876} C_VEL
LIN {X 0,Y 609.516,Z 1208.018,A -85,B 0,C 180,E1 28151.539,E2 28151.539} C_VEL
LIN {X 0,Y 610.489,Z 1194.96,A -85,B 0,C 180,E1 28149.077,E2 28149.077} C_VEL
LIN {X 0,Y 611.577,Z 1182.361,A -85,B 0,C 180,E1 28146.996,E2 28146.996} C_VEL
LIN {X 0,Y 612.925,Z 1168.147,A -85,B 0,C 180,E1 28144.9,E2 28144.9} C_VEL
LIN {X 0,Y 614.893,Z 1149.552,A -85,B 0,C 180,E1 28142.493,E2 28142.493} C_VEL
LIN {X 0,Y 616.618,Z 1133.736,A -85,B 0,C 180,E1 28140.675,E2 28140.675} C_VEL
LIN {X 0,Y 618.572,Z 1117.087,A -85,B 0,C 180,E1 28138.951,E2 28138.951} C_VEL
LIN {X 0,Y 621.234,Z 1095.147,A -85,B 0,C 180,E1 28136.93,E2 28136.93} C_VEL
LIN {X 0,Y 623.551,Z 1075.649,A -85,B 0,C 180,E1 28135.348,E2 28135.348} C_VEL
LIN {X 0,Y 625.781,Z 1056.858,A -85,B 0,C 180,E1 28133.982,E2 28133.982} C_VEL
LIN {X 0,Y 628.143,Z 1036.529,A -85,B 0,C 180,E1 28132.662,E2 28132.662} C_VEL
LIN {X 0,Y 631,Z 1010.52,A -85,B 0,C 180,E1 28131.195,E2 28131.195} C_VEL
LIN {X 0,Y 633.126,Z 989.51,A -85,B 0,C 180,E1 28130.176,E2 28130.176} C_VEL
LIN {X 0,Y 635.029,Z 969.185,A -85,B 0,C 180,E1 28129.315,E2 28129.315} C_VEL
LIN {X 0,Y 636.8,Z 948.432,A -85,B 0,C 180,E1 28128.558,E2 28128.558} C_VEL
LIN {X 0,Y 638.625,Z 924.317,A -85,B 0,C 180,E1 28127.819,E2 28127.819} C_VEL
LIN {X 0,Y 640.327,Z 896.028,A -85,B 0,C 180,E1 28127.15,E2 28127.15} C_VEL
LIN {X 0,Y 641.356,Z 873.072,A -85,B 0,C 180,E1 28126.747,E2 28126.747} C_VEL
LIN {X 0,Y 646.049,Z 660.635,A -85,B 0,C 180,E1 28123.861,E2 28123.861} C_VEL
LIN {X 0,Y 650.67,Z 461.379,A -85,B 0,C 180,E1 28121.097,E2 28121.097} C_VEL
LIN {X 0,Y 640.244,Z 446.803,A -85,B 0,C 180,E1 28119.757,E2 28119.757} C_VEL
LIN {X 0,Y 629.531,Z 432.563,A -85,B 0,C 180,E1 28118.305,E2 28118.305} C_VEL
LIN {X 0,Y 625.027,Z 426.866,A -85,B 0,C 180,E1 28117.67,E2 28117.67} C_VEL
LIN {X 0,Y 621.405,Z 422.166,A -85,B 0,C 180,E1 28117.143,E2 28117.143} C_VEL
LIN {X 0,Y 618.171,Z 417.822,A -85,B 0,C 180,E1 28116.66,E2 28116.66} C_VEL
LIN {X 0,Y 614.457,Z 413.596,A -85,B 0,C 180,E1 28116.106,E2 28116.106} C_VEL
LIN {X 0,Y 613.143,Z 411.37,A -85,B 0,C 180,E1 28115.892,E2 28115.892} C_VEL
LIN {X 0,Y 610.478,Z 408.989,A -85,B 0,C 180,E1 28115.495,E2 28115.495} C_VEL
LIN {X 0,Y 609.174,Z 405.986,A -85,B 0,C 180,E1 28115.261,E2 28115.261} C_VEL
LIN {X 0,Y 609.065,Z 405.331,A -85,B 0,C 180,E1 28115.222,E2 28115.222} C_VEL
LIN {X 0,Y 609.067,Z 405.356,A -85,B 0,C 180,E1 28111.912,E2 28111.912} C_VEL
LIN {X 0,Y 609.068,Z 405.349,A -85,B 0,C 180,E1 28108.752,E2 28108.752} C_VEL
LIN {X 0,Y 609.057,Z 405.324,A -85,B 0,C 180,E1 28105.58,E2 28105.58} C_VEL
LIN {X 0,Y 609.063,Z 405.357,A -85,B 0,C 180,E1 28102.388,E2 28102.388} C_VEL
LIN {X 0,Y 609.053,Z 405.338,A -85,B 0,C 180,E1 28099.265,E2 28099.265} C_VEL
LIN {X 0,Y 609.063,Z 405.34,A -85,B 0,C 180,E1 28096.108,E2 28096.108} C_VEL
LIN {X 0,Y 609.051,Z 405.351,A -85,B 0,C 180,E1 28092.998,E2 28092.998} C_VEL
LIN {X 0,Y 609.061,Z 405.329,A -85,B 0,C 180,E1 28089.831,E2 28089.831} C_VEL
LIN {X 0,Y 609.048,Z 405.356,A -85,B 0,C 180,E1 28086.656,E2 28086.656} C_VEL
LIN {X 0,Y 609.063,Z 405.324,A -85,B 0,C 180,E1 28083.577,E2 28083.577} C_VEL
LIN {X 0,Y 609.046,Z 405.358,A -85,B 0,C 180,E1 28080.376,E2 28080.376} C_VEL
LIN {X 0,Y 609.063,Z 405.319,A -85,B 0,C 180,E1 28077.271,E2 28077.271} C_VEL
LIN {X 0,Y 609.044,Z 405.359,A -85,B 0,C 180,E1 28074.158,E2 28074.158} C_VEL
LIN {X 0,Y 609.064,Z 405.319,A -85,B 0,C 180,E1 28071.027,E2 28071.027} C_VEL
LIN {X 0,Y 609.043,Z 405.364,A -85,B 0,C 180,E1 28067.869,E2 28067.869} C_VEL
LIN {X 0,Y 609.069,Z 405.324,A -85,B 0,C 180,E1 28064.674,E2 28064.674} C_VEL
LIN {X 0,Y 609.045,Z 405.357,A -85,B 0,C 180,E1 28061.527,E2 28061.527} C_VEL
LIN {X 0,Y 609.071,Z 405.348,A -85,B 0,C 180,E1 28058.222,E2 28058.222} C_VEL
LIN {X 0,Y 609.055,Z 405.329,A -85,B 0,C 180,E1 28055.044,E2 28055.044} C_VEL
LIN {X 0,Y 609.05,Z 405.357,A -85,B 0,C 180,E1 28051.783,E2 28051.783} C_VEL
LIN {X 0,Y 609.073,Z 405.355,A -85,B 0,C 180,E1 28048.615,E2 28048.615} C_VEL
LIN {X 0,Y 609.07,Z 405.437,A -85,B 0,C 180,E1 28046.728,E2 28046.728} C_VEL
LIN {X 0,Y 610.506,Z 409.002,A -85,B 0,C 180,E1 28046.161,E2 28046.161} C_VEL
LIN {X 0,Y 611.644,Z 410.911,A -85,B 0,C 180,E1 28045.813,E2 28045.813} C_VEL
LIN {X 0,Y 616.68,Z 420.957,A -85,B 0,C 180,E1 28044.167,E2 28044.167} C_VEL
LIN {X 0,Y 618.988,Z 425.343,A -85,B 0,C 180,E1 28043.512,E2 28043.512} C_VEL
LIN {X 0,Y 629.911,Z 440.488,A -85,B 0,C 180,E1 28041.925,E2 28041.925} C_VEL
LIN {X 0,Y 644.523,Z 461.56,A -85,B 0,C 180,E1 28039.952,E2 28039.952} C_VEL
LIN {X 0,Y 650.971,Z 471.498,A -85,B 0,C 180,E1 28039.123,E2 28039.123} C_VEL
LIN {X 0,Y 646.238,Z 679.539,A -85,B 0,C 180,E1 28036.241,E2 28036.241} C_VEL
LIN {X 0,Y 641.511,Z 898.786,A -85,B 0,C 180,E1 28033.272,E2 28033.272} C_VEL
LIN {X 0,Y 640.548,Z 921.513,A -85,B 0,C 180,E1 28032.892,E2 28032.892} C_VEL
LIN {X 0,Y 639.311,Z 943.411,A -85,B 0,C 180,E1 28032.414,E2 28032.414} C_VEL
LIN {X 0,Y 637.673,Z 967.737,A -85,B 0,C 180,E1 28031.746,E2 28031.746} C_VEL
LIN {X 0,Y 635.436,Z 994.836,A -85,B 0,C 180,E1 28030.81,E2 28030.81} C_VEL
LIN {X 0,Y 633.392,Z 1016.899,A -85,B 0,C 180,E1 28029.895,E2 28029.895} C_VEL
LIN {X 0,Y 631.305,Z 1037.634,A -85,B 0,C 180,E1 28028.905,E2 28028.905} C_VEL
LIN {X 0,Y 628.894,Z 1059.971,A -85,B 0,C 180,E1 28027.688,E2 28027.688} C_VEL
LIN {X 0,Y 626.019,Z 1084.805,A -85,B 0,C 180,E1 28026.115,E2 28026.115} C_VEL
LIN {X 0,Y 623.752,Z 1103.854,A -85,B 0,C 180,E1 28024.744,E2 28024.744} C_VEL
LIN {X 0,Y 621.566,Z 1122.226,A -85,B 0,C 180,E1 28023.271,E2 28023.271} C_VEL
LIN {X 0,Y 619.085,Z 1143.165,A -85,B 0,C 180,E1 28021.394,E2 28021.394} C_VEL
LIN {X 0,Y 616.766,Z 1162.419,A -85,B 0,C 180,E1 28019.424,E2 28019.424} C_VEL
LIN {X 0,Y 615.026,Z 1178.24,A -85,B 0,C 180,E1 28017.619,E2 28017.619} C_VEL
LIN {X 0,Y 613.186,Z 1195.738,A -85,B 0,C 180,E1 28015.394,E2 28015.394} C_VEL
LIN {X 0,Y 611.664,Z 1211.446,A -85,B 0,C 180,E1 28013.103,E2 28013.103} C_VEL
LIN {X 0,Y 610.547,Z 1224.167,A -85,B 0,C 180,E1 28011.014,E2 28011.014} C_VEL
LIN {X 0,Y 609.558,Z 1237.453,A -85,B 0,C 180,E1 28008.535,E2 28008.535} C_VEL
LIN {X 0,Y 608.902,Z 1248.426,A -85,B 0,C 180,E1 28006.128,E2 28006.128} C_VEL
LIN {X 0,Y 608.481,Z 1256.147,A -85,B 0,C 180,E1 28004.176,E2 28004.176} C_VEL
LIN {X 0,Y 608.236,Z 1262.738,A -85,B 0,C 180,E1 28002.247,E2 28002.247} C_VEL
LIN {X 0,Y 608.074,Z 1268.809,A -85,B 0,C 180,E1 28000.137,E2 28000.137} C_VEL
LIN {X 0,Y 607.943,Z 1274.339,A -85,B 0,C 180,E1 27997.755,E2 27997.755} C_VEL
LIN {X 0,Y 607.92,Z 1278.547,A -85,B 0,C 180,E1 27995.194,E2 27995.194} C_VEL
LIN {X 0,Y 607.91,Z 1280.741,A -85,B 0,C 180,E1 27993.021,E2 27993.021} C_VEL
LIN {X 0,Y 607.877,Z 1281.758,A -85,B 0,C 180,E1 27991.041,E2 27991.041} C_VEL
LIN {X 0,Y 607.866,Z 1281.806,A -85,B 0,C 180,E1 27989.156,E2 27989.156} C_VEL
LIN {X 0,Y 607.91,Z 1280.95,A -85,B 0,C 180,E1 27987.27,E2 27987.27} C_VEL
LIN {X 0,Y 607.916,Z 1279.012,A -85,B 0,C 180,E1 27985.193,E2 27985.193} C_VEL
LIN {X 0,Y 607.957,Z 1275.43,A -85,B 0,C 180,E1 27982.824,E2 27982.824} C_VEL
LIN {X 0,Y 608.01,Z 1270.104,A -85,B 0,C 180,E1 27980.348,E2 27980.348} C_VEL
LIN {X 0,Y 608.215,Z 1263.534,A -85,B 0,C 180,E1 27978.006,E2 27978.006} C_VEL
LIN {X 0,Y 608.442,Z 1256.884,A -85,B 0,C 180,E1 27976.026,E2 27976.026} C_VEL
LIN {X 0,Y 608.872,Z 1248.923,A -85,B 0,C 180,E1 27973.99,E2 27973.99} C_VEL
LIN {X 0,Y 609.448,Z 1239.021,A -85,B 0,C 180,E1 27971.794,E2 27971.794} C_VEL
LIN {X 0,Y 610.427,Z 1225.869,A -85,B 0,C 180,E1 27969.279,E2 27969.279} C_VEL
LIN {X 0,Y 611.54,Z 1212.775,A -85,B 0,C 180,E1 27967.105,E2 27967.105} C_VEL
LIN {X 0,Y 612.816,Z 1199.323,A -85,B 0,C 180,E1 27965.111,E2 27965.111} C_VEL
LIN {X 0,Y 614.658,Z 1181.802,A -85,B 0,C 180,E1 27962.805,E2 27962.805} C_VEL
LIN {X 0,Y 616.551,Z 1164.356,A -85,B 0,C 180,E1 27960.788,E2 27960.788} C_VEL
LIN {X 0,Y 618.366,Z 1148.762,A -85,B 0,C 180,E1 27959.163,E2 27959.163} C_VEL
LIN {X 0,Y 620.706,Z 1129.455,A -85,B 0,C 180,E1 27957.347,E2 27957.347} C_VEL
LIN {X 0,Y 623.363,Z 1107.309,A -85,B 0,C 180,E1 27955.52,E2 27955.52} C_VEL
LIN {X 0,Y 625.614,Z 1088.295,A -85,B 0,C 180,E1 27954.127,E2 27954.127} C_VEL
LIN {X 0,Y 627.827,Z 1069.281,A -85,B 0,C 180,E1 27952.879,E2 27952.879} C_VEL
LIN {X 0,Y 630.375,Z 1046.644,A -85,B 0,C 180,E1 27951.561,E2 27951.561} C_VEL
LIN {X 0,Y 632.973,Z 1021.098,A -85,B 0,C 180,E1 27950.292,E2 27950.292} C_VEL
LIN {X 0,Y 634.996,Z 999.552,A -85,B 0,C 180,E1 27949.374,E2 27949.374} C_VEL
LIN {X 0,Y 636.749,Z 979.072,A -85,B 0,C 180,E1 27948.625,E2 27948.625} C_VEL
LIN {X 0,Y 638.479,Z 956.276,A -85,B 0,C 180,E1 27947.921,E2 27947.921} C_VEL
LIN {X 0,Y 640.249,Z 927.773,A -85,B 0,C 180,E1 27947.23,E2 27947.23} C_VEL
LIN {X 0,Y 641.337,Z 903.647,A -85,B 0,C 180,E1 27946.801,E2 27946.801} C_VEL
LIN {X 0,Y 645.742,Z 702.684,A -85,B 0,C 180,E1 27944.075,E2 27944.075} C_VEL
LIN {X 0,Y 650.621,Z 486.659,A -85,B 0,C 180,E1 27941.09,E2 27941.09} C_VEL
LIN {X 0,Y 650.884,Z 471.1,A -85,B 0,C 180,E1 27940.862,E2 27940.862} C_VEL
LIN {X 0,Y 636.374,Z 449.732,A -85,B 0,C 180,E1 27938.968,E2 27938.968} C_VEL
LIN {X 0,Y 626.644,Z 435.96,A -85,B 0,C 180,E1 27937.613,E2 27937.613} C_VEL
LIN {X 0,Y 618.446,Z 424.425,A -85,B 0,C 180,E1 27936.386,E2 27936.386} C_VEL
LIN {X 0,Y 615.152,Z 418.008,A -85,B 0,C 180,E1 27935.356,E2 27935.356} C_VEL
LIN {X 0,Y 613.107,Z 413.968,A -85,B 0,C 180,E1 27934.693,E2 27934.693} C_VEL
LIN {X 0,Y 610.835,Z 409.418,A -85,B 0,C 180,E1 27933.931,E2 27933.931} C_VEL
LIN {X 0,Y 609.127,Z 405.969,A -85,B 0,C 180,E1 27933.342,E2 27933.342} C_VEL
LIN {X 0,Y 609.015,Z 405.338,A -85,B 0,C 180,E1 27933.255,E2 27933.255} C_VEL
LIN {X 0,Y 609.016,Z 405.338,A -85,B 0,C 180,E1 27930.478,E2 27930.478} C_VEL
LIN {X 0,Y 609.016,Z 405.366,A -85,B 0,C 180,E1 27927.157,E2 27927.157} C_VEL
LIN {X 0,Y 609.004,Z 405.342,A -85,B 0,C 180,E1 27924.337,E2 27924.337} C_VEL
LIN {X 0,Y 609.01,Z 405.338,A -85,B 0,C 180,E1 27921.073,E2 27921.073} C_VEL
LIN {X 0,Y 608.992,Z 405.366,A -85,B 0,C 180,E1 27918.276,E2 27918.276} C_VEL
LIN {X 0,Y 609.021,Z 405.328,A -85,B 0,C 180,E1 27915.132,E2 27915.132} C_VEL
LIN {X 0,Y 608.976,Z 405.371,A -85,B 0,C 180,E1 27912.325,E2 27912.325} C_VEL
LIN {X 0,Y 609.047,Z 405.324,A -85,B 0,C 180,E1 27909.259,E2 27909.259} C_VEL
LIN {X 0,Y 608.97,Z 405.372,A -85,B 0,C 180,E1 27906.316,E2 27906.316} C_VEL
LIN {X 0,Y 609.023,Z 405.327,A -85,B 0,C 180,E1 27903.388,E2 27903.388} C_VEL
LIN {X 0,Y 608.984,Z 405.371,A -85,B 0,C 180,E1 27900.282,E2 27900.282} C_VEL
LIN {X 0,Y 608.998,Z 405.333,A -85,B 0,C 180,E1 27897.553,E2 27897.553} C_VEL
LIN {X 0,Y 609.001,Z 405.369,A -85,B 0,C 180,E1 27894.252,E2 27894.252} C_VEL
LIN {X 0,Y 608.996,Z 405.335,A -85,B 0,C 180,E1 27891.597,E2 27891.597} C_VEL
LIN {X 0,Y 609.046,Z 405.367,A -85,B 0,C 180,E1 27888.446,E2 27888.446} C_VEL
LIN {X 0,Y 609.001,Z 405.333,A -85,B 0,C 180,E1 27885.548,E2 27885.548} C_VEL
LIN {X 0,Y 609.07,Z 405.364,A -85,B 0,C 180,E1 27882.418,E2 27882.418} C_VEL
LIN {X 0,Y 609.009,Z 405.328,A -85,B 0,C 180,E1 27879.43,E2 27879.43} C_VEL
LIN {X 0,Y 609.076,Z 405.356,A -85,B 0,C 180,E1 27876.335,E2 27876.335} C_VEL
LIN {X 0,Y 609.021,Z 405.344,A -85,B 0,C 180,E1 27873.254,E2 27873.254} C_VEL
LIN {X 0,Y 609.077,Z 405.326,A -85,B 0,C 180,E1 27870.17,E2 27870.17} C_VEL
LIN {X 0,Y 609.034,Z 405.361,A -85,B 0,C 180,E1 27867.015,E2 27867.015} C_VEL
LIN {X 0,Y 609.072,Z 405.506,A -85,B 0,C 180,E1 27864.668,E2 27864.668} C_VEL
LIN {X 0,Y 610.194,Z 408.545,A -85,B 0,C 180,E1 27864.457,E2 27864.457} C_VEL
LIN {X 0,Y 612.697,Z 411.093,A -85,B 0,C 180,E1 27864.078,E2 27864.078} C_VEL
LIN {X 0,Y 613.626,Z 412.02,A -85,B 0,C 180,E1 27863.939,E2 27863.939} C_VEL
LIN {X 0,Y 616.048,Z 415.756,A -85,B 0,C 180,E1 27863.555,E2 27863.555} C_VEL
LIN {X 0,Y 618.334,Z 418.121,A -85,B 0,C 180,E1 27863.221,E2 27863.221} C_VEL
LIN {X 0,Y 621.657,Z 422.375,A -85,B 0,C 180,E1 27862.73,E2 27862.73} C_VEL
LIN {X 0,Y 634.907,Z 439.581,A -85,B 0,C 180,E1 27860.867,E2 27860.867} C_VEL
LIN {X 0,Y 646.704,Z 455.715,A -85,B 0,C 180,E1 27859.316,E2 27859.316} C_VEL
LIN {X 0,Y 650.676,Z 461.711,A -85,B 0,C 180,E1 27858.807,E2 27858.807} C_VEL
LIN {X 0,Y 648.07,Z 571.425,A -85,B 0,C 180,E1 27857.278,E2 27857.278} C_VEL
LIN {X 0,Y 647.214,Z 579.129,A -85,B 0,C 180,E1 27857.237,E2 27857.237} C_VEL
LIN {X 0,Y 642.508,Z 599.798,A -85,B 0,C 180,E1 27857.36,E2 27857.36} C_VEL
LIN {X 0,Y 641.824,Z 606.408,A -85,B 0,C 180,E1 27857.32,E2 27857.32} C_VEL
LIN {X 0,Y 636.757,Z 824.386,A -85,B 0,C 180,E1 27854.332,E2 27854.332} C_VEL
LIN {X 0,Y 635.35,Z 878.086,A -85,B 0,C 180,E1 27853.582,E2 27853.582} C_VEL
LIN {X 0,Y 633.815,Z 906.846,A -85,B 0,C 180,E1 27853.019,E2 27853.019} C_VEL
LIN {X 0,Y 632.243,Z 929.545,A -85,B 0,C 180,E1 27852.43,E2 27852.43} C_VEL
LIN {X 0,Y 630.581,Z 950.195,A -85,B 0,C 180,E1 27851.779,E2 27851.779} C_VEL
LIN {X 0,Y 628.778,Z 970.057,A -85,B 0,C 180,E1 27851.045,E2 27851.045} C_VEL
LIN {X 0,Y 626.549,Z 992.524,A -85,B 0,C 180,E1 27850.077,E2 27850.077} C_VEL
LIN {X 0,Y 623.684,Z 1018.654,A -85,B 0,C 180,E1 27848.751,E2 27848.751} C_VEL
LIN {X 0,Y 621.209,Z 1039.461,A -85,B 0,C 180,E1 27847.526,E2 27847.526} C_VEL
LIN {X 0,Y 618.861,Z 1058.433,A -85,B 0,C 180,E1 27846.27,E2 27846.27} C_VEL
LIN {X 0,Y 616.319,Z 1078.778,A -85,B 0,C 180,E1 27844.761,E2 27844.761} C_VEL
LIN {X 0,Y 613.343,Z 1101.78,A -85,B 0,C 180,E1 27842.816,E2 27842.816} C_VEL
LIN {X 0,Y 611.127,Z 1119.098,A -85,B 0,C 180,E1 27841.162,E2 27841.162} C_VEL
LIN {X 0,Y 609.104,Z 1135.357,A -85,B 0,C 180,E1 27839.442,E2 27839.442} C_VEL
LIN {X 0,Y 606.953,Z 1153.901,A -85,B 0,C 180,E1 27837.25,E2 27837.25} C_VEL
LIN {X 0,Y 605.097,Z 1170.423,A -85,B 0,C 180,E1 27835.019,E2 27835.019} C_VEL
LIN {X 0,Y 603.721,Z 1184.1,A -85,B 0,C 180,E1 27832.948,E2 27832.948} C_VEL
LIN {X 0,Y 602.392,Z 1198.952,A -85,B 0,C 180,E1 27830.394,E2 27830.394} C_VEL
LIN {X 0,Y 601.488,Z 1210.436,A -85,B 0,C 180,E1 27828.105,E2 27828.105} C_VEL
LIN {X 0,Y 600.897,Z 1219.952,A -85,B 0,C 180,E1 27825.93,E2 27825.93} C_VEL
LIN {X 0,Y 600.422,Z 1228.84,A -85,B 0,C 180,E1 27823.575,E2 27823.575} C_VEL
LIN {X 0,Y 600.133,Z 1236.927,A -85,B 0,C 180,E1 27820.944,E2 27820.944} C_VEL
LIN {X 0,Y 600.005,Z 1242.639,A -85,B 0,C 180,E1 27818.621,E2 27818.621} C_VEL
LIN {X 0,Y 599.943,Z 1247.12,A -85,B 0,C 180,E1 27816.214,E2 27816.214} C_VEL
LIN {X 0,Y 599.914,Z 1250.306,A -85,B 0,C 180,E1 27813.627,E2 27813.627} C_VEL
LIN {X 0,Y 599.896,Z 1251.704,A -85,B 0,C 180,E1 27811.237,E2 27811.237} C_VEL
LIN {X 0,Y 599.864,Z 1251.836,A -85,B 0,C 180,E1 27809.232,E2 27809.232} C_VEL
LIN {X 0,Y 599.909,Z 1250.976,A -85,B 0,C 180,E1 27807.225,E2 27807.225} C_VEL
LIN {X 0,Y 599.916,Z 1249.053,A -85,B 0,C 180,E1 27805.12,E2 27805.12} C_VEL
LIN {X 0,Y 599.958,Z 1245.496,A -85,B 0,C 180,E1 27802.719,E2 27802.719} C_VEL
LIN {X 0,Y 600.026,Z 1240.198,A -85,B 0,C 180,E1 27800.21,E2 27800.21} C_VEL
LIN {X 0,Y 600.246,Z 1233.483,A -85,B 0,C 180,E1 27797.783,E2 27797.783} C_VEL
LIN {X 0,Y 600.518,Z 1226.591,A -85,B 0,C 180,E1 27795.711,E2 27795.711} C_VEL
LIN {X 0,Y 600.976,Z 1218.662,A -85,B 0,C 180,E1 27793.666,E2 27793.666} C_VEL
LIN {X 0,Y 601.661,Z 1208.016,A -85,B 0,C 180,E1 27791.289,E2 27791.289} C_VEL
LIN {X 0,Y 602.707,Z 1194.954,A -85,B 0,C 180,E1 27788.794,E2 27788.794} C_VEL
LIN {X 0,Y 603.886,Z 1182.355,A -85,B 0,C 180,E1 27786.685,E2 27786.685} C_VEL
LIN {X 0,Y 605.336,Z 1168.145,A -85,B 0,C 180,E1 27784.563,E2 27784.563} C_VEL
LIN {X 0,Y 607.441,Z 1149.513,A -85,B 0,C 180,E1 27782.122,E2 27782.122} C_VEL
LIN {X 0,Y 609.297,Z 1133.729,A -85,B 0,C 180,E1 27780.288,E2 27780.288} C_VEL
LIN {X 0,Y 611.391,Z 1117.134,A -85,B 0,C 180,E1 27778.55,E2 27778.55} C_VEL
LIN {X 0,Y 614.159,Z 1095.745,A -85,B 0,C 180,E1 27776.555,E2 27776.555} C_VEL
LIN {X 0,Y 616.675,Z 1075.717,A -85,B 0,C 180,E1 27774.912,E2 27774.912} C_VEL
LIN {X 0,Y 619.058,Z 1056.846,A -85,B 0,C 180,E1 27773.528,E2 27773.528} C_VEL
LIN {X 0,Y 621.629,Z 1035.992,A -85,B 0,C 180,E1 27772.165,E2 27772.165} C_VEL
LIN {X 0,Y 624.621,Z 1010.403,A -85,B 0,C 180,E1 27770.717,E2 27770.717} C_VEL
LIN {X 0,Y 626.905,Z 989.039,A -85,B 0,C 180,E1 27769.676,E2 27769.676} C_VEL
LIN {X 0,Y 628.988,Z 967.88,A -85,B 0,C 180,E1 27768.78,E2 27768.78} C_VEL
LIN {X 0,Y 630.866,Z 946.877,A -85,B 0,C 180,E1 27768.017,E2 27768.017} C_VEL
LIN {X 0,Y 632.966,Z 920.346,A -85,B 0,C 180,E1 27767.22,E2 27767.22} C_VEL
LIN {X 0,Y 634.518,Z 894.508,A -85,B 0,C 180,E1 27766.627,E2 27766.627} C_VEL
LIN {X 0,Y 635.547,Z 872.45,A -85,B 0,C 180,E1 27766.242,E2 27766.242} C_VEL
LIN {X 0,Y 640.523,Z 660.755,A -85,B 0,C 180,E1 27763.343,E2 27763.343} C_VEL
LIN {X 0,Y 645.336,Z 465.335,A -85,B 0,C 180,E1 27760.614,E2 27760.614} C_VEL
LIN {X 0,Y 633.274,Z 448.658,A -85,B 0,C 180,E1 27759.02,E2 27759.02} C_VEL
LIN {X 0,Y 622.341,Z 434.205,A -85,B 0,C 180,E1 27757.483,E2 27757.483} C_VEL
LIN {X 0,Y 617.523,Z 428.192,A -85,B 0,C 180,E1 27756.777,E2 27756.777} C_VEL
LIN {X 0,Y 613.982,Z 423.571,A -85,B 0,C 180,E1 27756.239,E2 27756.239} C_VEL
LIN {X 0,Y 610.672,Z 419.376,A -85,B 0,C 180,E1 27755.727,E2 27755.727} C_VEL
LIN {X 0,Y 609.577,Z 418.009,A -85,B 0,C 180,E1 27755.555,E2 27755.555} C_VEL
LIN {X 0,Y 606.61,Z 414.61,A -85,B 0,C 180,E1 27755.09,E2 27755.09} C_VEL
LIN {X 0,Y 605.537,Z 412.511,A -85,B 0,C 180,E1 27754.901,E2 27754.901} C_VEL
LIN {X 0,Y 602.664,Z 410.135,A -85,B 0,C 180,E1 27754.455,E2 27754.455} C_VEL
LIN {X 0,Y 601.283,Z 407.165,A -85,B 0,C 180,E1 27754.199,E2 27754.199} C_VEL
LIN {X 0,Y 601.129,Z 406.315,A -85,B 0,C 180,E1 27754.134,E2 27754.134} C_VEL
LIN {X 0,Y 601.127,Z 406.316,A -85,B 0,C 180,E1 27750.872,E2 27750.872} C_VEL
LIN {X 0,Y 601.125,Z 406.353,A -85,B 0,C 180,E1 27747.651,E2 27747.651} C_VEL
LIN {X 0,Y 601.123,Z 406.323,A -85,B 0,C 180,E1 27744.468,E2 27744.468} C_VEL
LIN {X 0,Y 601.114,Z 406.323,A -85,B 0,C 180,E1 27741.327,E2 27741.327} C_VEL
LIN {X 0,Y 601.126,Z 406.35,A -85,B 0,C 180,E1 27738.123,E2 27738.123} C_VEL
LIN {X 0,Y 601.107,Z 406.311,A -85,B 0,C 180,E1 27734.941,E2 27734.941} C_VEL
LIN {X 0,Y 601.126,Z 406.352,A -85,B 0,C 180,E1 27731.806,E2 27731.806} C_VEL
LIN {X 0,Y 601.106,Z 406.308,A -85,B 0,C 180,E1 27728.61,E2 27728.61} C_VEL
LIN {X 0,Y 601.13,Z 406.348,A -85,B 0,C 180,E1 27725.44,E2 27725.44} C_VEL
LIN {X 0,Y 601.111,Z 406.308,A -85,B 0,C 180,E1 27722.193,E2 27722.193} C_VEL
LIN {X 0,Y 601.134,Z 406.344,A -85,B 0,C 180,E1 27718.952,E2 27718.952} C_VEL
LIN {X 0,Y 601.124,Z 406.311,A -85,B 0,C 180,E1 27715.707,E2 27715.707} C_VEL
LIN {X 0,Y 601.113,Z 406.34,A -85,B 0,C 180,E1 27712.449,E2 27712.449} C_VEL
LIN {X 0,Y 601.13,Z 406.326,A -85,B 0,C 180,E1 27709.263,E2 27709.263} C_VEL
LIN {X 0,Y 601.101,Z 406.324,A -85,B 0,C 180,E1 27706.043,E2 27706.043} C_VEL
LIN {X 0,Y 601.133,Z 406.348,A -85,B 0,C 180,E1 27702.878,E2 27702.878} C_VEL
LIN {X 0,Y 601.097,Z 406.314,A -85,B 0,C 180,E1 27699.752,E2 27699.752} C_VEL
LIN {X 0,Y 601.134,Z 406.345,A -85,B 0,C 180,E1 27696.662,E2 27696.662} C_VEL
LIN {X 0,Y 601.1,Z 406.334,A -85,B 0,C 180,E1 27693.502,E2 27693.502} C_VEL
LIN {X 0,Y 601.133,Z 406.313,A -85,B 0,C 180,E1 27690.395,E2 27690.395} C_VEL
LIN {X 0,Y 601.142,Z 406.519,A -85,B 0,C 180,E1 27687.729,E2 27687.729} C_VEL
LIN {X 0,Y 602.265,Z 409.612,A -85,B 0,C 180,E1 27687.232,E2 27687.232} C_VEL
LIN {X 0,Y 603.602,Z 411.319,A -85,B 0,C 180,E1 27686.862,E2 27686.862} C_VEL
LIN {X 0,Y 605.493,Z 415.278,A -85,B 0,C 180,E1 27686.185,E2 27686.185} C_VEL
LIN {X 0,Y 610.427,Z 424.687,A -85,B 0,C 180,E1 27684.617,E2 27684.617} C_VEL
LIN {X 0,Y 625.421,Z 445.46,A -85,B 0,C 180,E1 27682.358,E2 27682.358} C_VEL
LIN {X 0,Y 641.562,Z 469.029,A -85,B 0,C 180,E1 27680.138,E2 27680.138} C_VEL
LIN {X 0,Y 645.614,Z 475.446,A -85,B 0,C 180,E1 27679.605,E2 27679.605} C_VEL
LIN {X 0,Y 640.576,Z 684.149,A -85,B 0,C 180,E1 27676.695,E2 27676.695} C_VEL
LIN {X 0,Y 635.621,Z 900.522,A -85,B 0,C 180,E1 27673.741,E2 27673.741} C_VEL
LIN {X 0,Y 634.632,Z 922.3,A -85,B 0,C 180,E1 27673.371,E2 27673.371} C_VEL
LIN {X 0,Y 633.327,Z 944.13,A -85,B 0,C 180,E1 27672.889,E2 27672.889} C_VEL
LIN {X 0,Y 631.486,Z 970.127,A -85,B 0,C 180,E1 27672.163,E2 27672.163} C_VEL
LIN {X 0,Y 629.207,Z 995.642,A -85,B 0,C 180,E1 27671.263,E2 27671.263} C_VEL
LIN {X 0,Y 627.193,Z 1016.383,A -85,B 0,C 180,E1 27670.398,E2 27670.398} C_VEL
LIN {X 0,Y 625.154,Z 1035.62,A -85,B 0,C 180,E1 27669.48,E2 27669.48} C_VEL
LIN {X 0,Y 623,Z 1054.578,A -85,B 0,C 180,E1 27668.459,E2 27668.459} C_VEL
LIN {X 0,Y 620.676,Z 1074.004,A -85,B 0,C 180,E1 27667.284,E2 27667.284} C_VEL
LIN {X 0,Y 617.715,Z 1097.844,A -85,B 0,C 180,E1 27665.645,E2 27665.645} C_VEL
LIN {X 0,Y 614.972,Z 1118.896,A -85,B 0,C 180,E1 27663.981,E2 27663.981} C_VEL
LIN {X 0,Y 612.787,Z 1136.013,A -85,B 0,C 180,E1 27662.471,E2 27662.471} C_VEL
LIN {X 0,Y 610.545,Z 1154.042,A -85,B 0,C 180,E1 27660.706,E2 27660.706} C_VEL
LIN {X 0,Y 608.071,Z 1174.117,A -85,B 0,C 180,E1 27658.484,E2 27658.484} C_VEL
LIN {X 0,Y 606.255,Z 1189.589,A -85,B 0,C 180,E1 27656.552,E2 27656.552} C_VEL
LIN {X 0,Y 604.64,Z 1204.863,A -85,B 0,C 180,E1 27654.423,E2 27654.423} C_VEL
LIN {X 0,Y 603.098,Z 1220.678,A -85,B 0,C 180,E1 27651.906,E2 27651.906} C_VEL
LIN {X 0,Y 602.128,Z 1232.252,A -85,B 0,C 180,E1 27649.805,E2 27649.805} C_VEL
LIN {X 0,Y 601.344,Z 1242.89,A -85,B 0,C 180,E1 27647.619,E2 27647.619} C_VEL
LIN {X 0,Y 600.695,Z 1254.005,A -85,B 0,C 180,E1 27644.955,E2 27644.955} C_VEL
LIN {X 0,Y 600.302,Z 1262.129,A -85,B 0,C 180,E1 27642.607,E2 27642.607} C_VEL
LIN {X 0,Y 600.113,Z 1268.046,A -85,B 0,C 180,E1 27640.565,E2 27640.565} C_VEL
LIN {X 0,Y 599.991,Z 1273.336,A -85,B 0,C 180,E1 27638.34,E2 27638.34} C_VEL
LIN {X 0,Y 599.934,Z 1277.776,A -85,B 0,C 180,E1 27635.839,E2 27635.839} C_VEL
LIN {X 0,Y 599.911,Z 1280.537,A -85,B 0,C 180,E1 27633.348,E2 27633.348} C_VEL
LIN {X 0,Y 599.892,Z 1281.713,A -85,B 0,C 180,E1 27631.246,E2 27631.246} C_VEL
LIN {X 0,Y 599.864,Z 1281.828,A -85,B 0,C 180,E1 27629.24,E2 27629.24} C_VEL
LIN {X 0,Y 599.91,Z 1280.951,A -85,B 0,C 180,E1 27627.234,E2 27627.234} C_VEL
LIN {X 0,Y 599.918,Z 1279.009,A -85,B 0,C 180,E1 27625.129,E2 27625.129} C_VEL
LIN {X 0,Y 599.956,Z 1275.431,A -85,B 0,C 180,E1 27622.728,E2 27622.728} C_VEL
LIN {X 0,Y 600.03,Z 1270.103,A -85,B 0,C 180,E1 27620.219,E2 27620.219} C_VEL
LIN {X 0,Y 600.237,Z 1263.673,A -85,B 0,C 180,E1 27617.889,E2 27617.889} C_VEL
LIN {X 0,Y 600.499,Z 1256.883,A -85,B 0,C 180,E1 27615.837,E2 27615.837} C_VEL
LIN {X 0,Y 600.962,Z 1248.921,A -85,B 0,C 180,E1 27613.774,E2 27613.774} C_VEL
LIN {X 0,Y 601.567,Z 1239.25,A -85,B 0,C 180,E1 27611.596,E2 27611.596} C_VEL
LIN {X 0,Y 602.634,Z 1225.904,A -85,B 0,C 180,E1 27609.005,E2 27609.005} C_VEL
LIN {X 0,Y 603.857,Z 1212.666,A -85,B 0,C 180,E1 27606.78,E2 27606.78} C_VEL
LIN {X 0,Y 605.287,Z 1198.615,A -85,B 0,C 180,E1 27604.675,E2 27604.675} C_VEL
LIN {X 0,Y 607.384,Z 1180.11,A -85,B 0,C 180,E1 27602.239,E2 27602.239} C_VEL
LIN {X 0,Y 609.268,Z 1163.975,A -85,B 0,C 180,E1 27600.36,E2 27600.36} C_VEL
LIN {X 0,Y 611.356,Z 1147.398,A -85,B 0,C 180,E1 27598.622,E2 27598.622} C_VEL
LIN {X 0,Y 614.089,Z 1126.298,A -85,B 0,C 180,E1 27596.647,E2 27596.647} C_VEL
LIN {X 0,Y 616.653,Z 1105.879,A -85,B 0,C 180,E1 27594.97,E2 27594.97} C_VEL
LIN {X 0,Y 619.028,Z 1087.058,A -85,B 0,C 180,E1 27593.589,E2 27593.589} C_VEL
LIN {X 0,Y 621.619,Z 1066.033,A -85,B 0,C 180,E1 27592.212,E2 27592.212} C_VEL
LIN {X 0,Y 624.575,Z 1040.833,A -85,B 0,C 180,E1 27590.784,E2 27590.784} C_VEL
LIN {X 0,Y 626.926,Z 1018.854,A -85,B 0,C 180,E1 27589.712,E2 27589.712} C_VEL
LIN {X 0,Y 628.931,Z 998.445,A -85,B 0,C 180,E1 27588.847,E2 27588.847} C_VEL
LIN {X 0,Y 630.801,Z 977.59,A -85,B 0,C 180,E1 27588.086,E2 27588.086} C_VEL
LIN {X 0,Y 632.868,Z 951.756,A -85,B 0,C 180,E1 27587.301,E2 27587.301} C_VEL
LIN {X 0,Y 634.496,Z 925.052,A -85,B 0,C 180,E1 27586.683,E2 27586.683} C_VEL
LIN {X 0,Y 635.537,Z 902.757,A -85,B 0,C 180,E1 27586.292,E2 27586.292} C_VEL
LIN {X 0,Y 640.288,Z 696.766,A -85,B 0,C 180,E1 27583.479,E2 27583.479} C_VEL
LIN {X 0,Y 645.413,Z 483.582,A -85,B 0,C 180,E1 27580.51,E2 27580.51} C_VEL
LIN {X 0,Y 645.456,Z 474.962,A -85,B 0,C 180,E1 27580.371,E2 27580.371} C_VEL
LIN {X 0,Y 629.085,Z 450.592,A -85,B 0,C 180,E1 27578.163,E2 27578.163} C_VEL
LIN {X 0,Y 617.143,Z 434.048,A -85,B 0,C 180,E1 27576.427,E2 27576.427} C_VEL
LIN {X 0,Y 609.769,Z 423.827,A -85,B 0,C 180,E1 27575.254,E2 27575.254} C_VEL
LIN {X 0,Y 605.478,Z 415.249,A -85,B 0,C 180,E1 27573.816,E2 27573.816} C_VEL
LIN {X 0,Y 603.563,Z 411.33,A -85,B 0,C 180,E1 27573.141,E2 27573.141} C_VEL
LIN {X 0,Y 601.453,Z 407.936,A -85,B 0,C 180,E1 27572.478,E2 27572.478} C_VEL
LIN {X 0,Y 601.112,Z 406.347,A -85,B 0,C 180,E1 27572.217,E2 27572.217} C_VEL
LIN {X 0,Y 601.067,Z 406.326,A -85,B 0,C 180,E1 27569.062,E2 27569.062} C_VEL
LIN {X 0,Y 601.079,Z 406.33,A -85,B 0,C 180,E1 27566.263,E2 27566.263} C_VEL
LIN {X 0,Y 601.069,Z 406.361,A -85,B 0,C 180,E1 27563.012,E2 27563.012} C_VEL
LIN {X 0,Y 601.058,Z 406.318,A -85,B 0,C 180,E1 27560.244,E2 27560.244} C_VEL
LIN {X 0,Y 601.063,Z 406.354,A -85,B 0,C 180,E1 27556.925,E2 27556.925} C_VEL
LIN {X 0,Y 601.042,Z 406.324,A -85,B 0,C 180,E1 27554.155,E2 27554.155} C_VEL
LIN {X 0,Y 601.067,Z 406.346,A -85,B 0,C 180,E1 27550.932,E2 27550.932} C_VEL
LIN {X 0,Y 601.029,Z 406.331,A -85,B 0,C 180,E1 27548.129,E2 27548.129} C_VEL
LIN {X 0,Y 601.101,Z 406.342,A -85,B 0,C 180,E1 27545.058,E2 27545.058} C_VEL
LIN {X 0,Y 601.035,Z 406.333,A -85,B 0,C 180,E1 27542.002,E2 27542.002} C_VEL
LIN {X 0,Y 601.12,Z 406.339,A -85,B 0,C 180,E1 27538.952,E2 27538.952} C_VEL
LIN {X 0,Y 601.045,Z 406.331,A -85,B 0,C 180,E1 27535.898,E2 27535.898} C_VEL
LIN {X 0,Y 601.139,Z 406.336,A -85,B 0,C 180,E1 27532.834,E2 27532.834} C_VEL
LIN {X 0,Y 601.056,Z 406.333,A -85,B 0,C 180,E1 27529.747,E2 27529.747} C_VEL
LIN {X 0,Y 601.135,Z 406.331,A -85,B 0,C 180,E1 27526.632,E2 27526.632} C_VEL
LIN {X 0,Y 601.067,Z 406.341,A -85,B 0,C 180,E1 27523.573,E2 27523.573} C_VEL
LIN {X 0,Y 601.135,Z 406.317,A -85,B 0,C 180,E1 27520.468,E2 27520.468} C_VEL
LIN {X 0,Y 601.078,Z 406.354,A -85,B 0,C 180,E1 27517.385,E2 27517.385} C_VEL
LIN {X 0,Y 601.133,Z 406.312,A -85,B 0,C 180,E1 27514.27,E2 27514.27} C_VEL
LIN {X 0,Y 601.087,Z 406.343,A -85,B 0,C 180,E1 27511.157,E2 27511.157} C_VEL
LIN {X 0,Y 601.135,Z 406.34,A -85,B 0,C 180,E1 27508.014,E2 27508.014} C_VEL
LIN {X 0,Y 601.155,Z 406.564,A -85,B 0,C 180,E1 27505.735,E2 27505.735} C_VEL
LIN {X 0,Y 602.253,Z 409.565,A -85,B 0,C 180,E1 27505.518,E2 27505.518} C_VEL
LIN {X 0,Y 604.821,Z 412.135,A -85,B 0,C 180,E1 27505.109,E2 27505.109} C_VEL
LIN {X 0,Y 605.798,Z 413.033,A -85,B 0,C 180,E1 27504.958,E2 27504.958} C_VEL
LIN {X 0,Y 608.22,Z 416.749,A -85,B 0,C 180,E1 27504.556,E2 27504.556} C_VEL
LIN {X 0,Y 610.452,Z 419.023,A -85,B 0,C 180,E1 27504.215,E2 27504.215} C_VEL
LIN {X 0,Y 613.68,Z 423.314,A -85,B 0,C 180,E1 27503.711,E2 27503.711} C_VEL
LIN {X 0,Y 615.522,Z 425.572,A -85,B 0,C 180,E1 27503.432,E2 27503.432} C_VEL
LIN {X 0,Y 620.163,Z 431.51,A -85,B 0,C 180,E1 27502.741,E2 27502.741} C_VEL
LIN {X 0,Y 628.428,Z 442.208,A -85,B 0,C 180,E1 27501.558,E2 27501.558} C_VEL
LIN {X 0,Y 641.482,Z 459.825,A -85,B 0,C 180,E1 27499.796,E2 27499.796} C_VEL
LIN {X 0,Y 645.338,Z 465.601,A -85,B 0,C 180,E1 27499.292,E2 27499.292} C_VEL
LIN {X 0,Y 641.824,Z 606.408,A -85,B 0,C 180,E1 27497.32,E2 27497.32} C_VEL
LIN {X 0,Y 640.946,Z 614.114,A -85,B 0,C 180,E1 27497.28,E2 27497.28} C_VEL
LIN {X 0,Y 636.22,Z 634.779,A -85,B 0,C 180,E1 27497.407,E2 27497.407} C_VEL
LIN {X 0,Y 635.541,Z 641.388,A -85,B 0,C 180,E1 27497.366,E2 27497.366} C_VEL
LIN {X 0,Y 630.053,Z 865.706,A -85,B 0,C 180,E1 27494.276,E2 27494.276} C_VEL
LIN {X 0,Y 628.936,Z 890.235,A -85,B 0,C 180,E1 27493.872,E2 27493.872} C_VEL
LIN {X 0,Y 627.626,Z 911.414,A -85,B 0,C 180,E1 27493.412,E2 27493.412} C_VEL
LIN {X 0,Y 626.017,Z 933.071,A -85,B 0,C 180,E1 27492.827,E2 27492.827} C_VEL
LIN {X 0,Y 623.976,Z 956.866,A -85,B 0,C 180,E1 27492.045,E2 27492.045} C_VEL
LIN {X 0,Y 621.315,Z 983.494,A -85,B 0,C 180,E1 27490.971,E2 27490.971} C_VEL
LIN {X 0,Y 619.015,Z 1004.052,A -85,B 0,C 180,E1 27489.999,E2 27489.999} C_VEL
LIN {X 0,Y 616.719,Z 1023.16,A -85,B 0,C 180,E1 27488.973,E2 27488.973} C_VEL
LIN {X 0,Y 614.252,Z 1042.712,A -85,B 0,C 180,E1 27487.79,E2 27487.79} C_VEL
LIN {X 0,Y 611.406,Z 1064.629,A -85,B 0,C 180,E1 27486.292,E2 27486.292} C_VEL
LIN {X 0,Y 608.24,Z 1087.593,A -85,B 0,C 180,E1 27484.487,E2 27484.487} C_VEL
LIN {X 0,Y 605.847,Z 1105.115,A -85,B 0,C 180,E1 27482.936,E2 27482.936} C_VEL
LIN {X 0,Y 603.517,Z 1122.481,A -85,B 0,C 180,E1 27481.229,E2 27481.229} C_VEL
LIN {X 0,Y 600.863,Z 1142.99,A -85,B 0,C 180,E1 27478.956,E2 27478.956} C_VEL
LIN {X 0,Y 598.875,Z 1158.563,A -85,B 0,C 180,E1 27477.003,E2 27477.003} C_VEL
LIN {X 0,Y 597.277,Z 1172.526,A -85,B 0,C 180,E1 27475.052,E2 27475.052} C_VEL
LIN {X 0,Y 595.634,Z 1188.232,A -85,B 0,C 180,E1 27472.588,E2 27472.588} C_VEL
LIN {X 0,Y 594.371,Z 1201.579,A -85,B 0,C 180,E1 27470.164,E2 27470.164} C_VEL
LIN {X 0,Y 593.527,Z 1211.813,A -85,B 0,C 180,E1 27468.052,E2 27468.052} C_VEL
LIN {X 0,Y 592.86,Z 1221.978,A -85,B 0,C 180,E1 27465.65,E2 27465.65} C_VEL
LIN {X 0,Y 592.386,Z 1231.405,A -85,B 0,C 180,E1 27462.968,E2 27462.968} C_VEL
LIN {X 0,Y 592.134,Z 1237.698,A -85,B 0,C 180,E1 27460.798,E2 27460.798} C_VEL
LIN {X 0,Y 592.011,Z 1243.05,A -85,B 0,C 180,E1 27458.543,E2 27458.543} C_VEL
LIN {X 0,Y 591.938,Z 1247.572,A -85,B 0,C 180,E1 27456.007,E2 27456.007} C_VEL
LIN {X 0,Y 591.912,Z 1250.443,A -85,B 0,C 180,E1 27453.482,E2 27453.482} C_VEL
LIN {X 0,Y 591.897,Z 1251.704,A -85,B 0,C 180,E1 27451.254,E2 27451.254} C_VEL
LIN {X 0,Y 591.864,Z 1251.836,A -85,B 0,C 180,E1 27449.221,E2 27449.221} C_VEL
LIN {X 0,Y 591.909,Z 1250.976,A -85,B 0,C 180,E1 27447.188,E2 27447.188} C_VEL
LIN {X 0,Y 591.918,Z 1249.049,A -85,B 0,C 180,E1 27445.054,E2 27445.054} C_VEL
LIN {X 0,Y 591.959,Z 1245.655,A -85,B 0,C 180,E1 27442.718,E2 27442.718} C_VEL
LIN {X 0,Y 592.035,Z 1240.45,A -85,B 0,C 180,E1 27440.175,E2 27440.175} C_VEL
LIN {X 0,Y 592.266,Z 1233.783,A -85,B 0,C 180,E1 27437.714,E2 27437.714} C_VEL
LIN {X 0,Y 592.583,Z 1226.657,A -85,B 0,C 180,E1 27435.535,E2 27435.535} C_VEL
LIN {X 0,Y 593.062,Z 1218.658,A -85,B 0,C 180,E1 27433.442,E2 27433.442} C_VEL
LIN {X 0,Y 593.777,Z 1208.48,A -85,B 0,C 180,E1 27431.133,E2 27431.133} C_VEL
LIN {X 0,Y 594.941,Z 1194.948,A -85,B 0,C 180,E1 27428.504,E2 27428.504} C_VEL
LIN {X 0,Y 596.199,Z 1182.349,A -85,B 0,C 180,E1 27426.367,E2 27426.367} C_VEL
LIN {X 0,Y 597.686,Z 1168.853,A -85,B 0,C 180,E1 27424.32,E2 27424.32} C_VEL
LIN {X 0,Y 599.916,Z 1150.34,A -85,B 0,C 180,E1 27421.848,E2 27421.848} C_VEL
LIN {X 0,Y 601.972,Z 1134.05,A -85,B 0,C 180,E1 27419.928,E2 27419.928} C_VEL
LIN {X 0,Y 604.173,Z 1117.633,A -85,B 0,C 180,E1 27418.187,E2 27418.187} C_VEL
LIN {X 0,Y 607.033,Z 1096.948,A -85,B 0,C 180,E1 27416.223,E2 27416.223} C_VEL
LIN {X 0,Y 609.847,Z 1075.706,A -85,B 0,C 180,E1 27414.46,E2 27414.46} C_VEL
LIN {X 0,Y 612.378,Z 1056.834,A -85,B 0,C 180,E1 27413.065,E2 27413.065} C_VEL
LIN {X 0,Y 615.145,Z 1035.69,A -85,B 0,C 180,E1 27411.673,E2 27411.673} C_VEL
LIN {X 0,Y 618.277,Z 1010.387,A -85,B 0,C 180,E1 27410.235,E2 27410.235} C_VEL
LIN {X 0,Y 620.682,Z 989.079,A -85,B 0,C 180,E1 27409.19,E2 27409.19} C_VEL
LIN {X 0,Y 622.811,Z 968.492,A -85,B 0,C 180,E1 27408.31,E2 27408.31} C_VEL
LIN {X 0,Y 624.793,Z 947.513,A -85,B 0,C 180,E1 27407.542,E2 27407.542} C_VEL
LIN {X 0,Y 626.925,Z 922.083,A -85,B 0,C 180,E1 27406.765,E2 27406.765} C_VEL
LIN {X 0,Y 628.655,Z 895.386,A -85,B 0,C 180,E1 27406.14,E2 27406.14} C_VEL
LIN {X 0,Y 629.759,Z 873.128,A -85,B 0,C 180,E1 27405.746,E2 27405.746} C_VEL
LIN {X 0,Y 634.941,Z 665.276,A -85,B 0,C 180,E1 27402.877,E2 27402.877} C_VEL
LIN {X 0,Y 640.036,Z 469.394,A -85,B 0,C 180,E1 27400.123,E2 27400.123} C_VEL
LIN {X 0,Y 626.82,Z 451.087,A -85,B 0,C 180,E1 27398.326,E2 27398.326} C_VEL
LIN {X 0,Y 614.87,Z 435.51,A -85,B 0,C 180,E1 27396.584,E2 27396.584} C_VEL
LIN {X 0,Y 610.157,Z 429.663,A -85,B 0,C 180,E1 27395.863,E2 27395.863} C_VEL
LIN {X 0,Y 606.312,Z 424.709,A -85,B 0,C 180,E1 27395.254,E2 27395.254} C_VEL
LIN {X 0,Y 603.017,Z 420.606,A -85,B 0,C 180,E1 27394.721,E2 27394.721} C_VEL
LIN {X 0,Y 602.024,Z 419.243,A -85,B 0,C 180,E1 27394.555,E2 27394.555} C_VEL
LIN {X 0,Y 598.99,Z 415.992,A -85,B 0,C 180,E1 27394.059,E2 27394.059} C_VEL
LIN {X 0,Y 597.579,Z 413.495,A -85,B 0,C 180,E1 27393.804,E2 27393.804} C_VEL
LIN {X 0,Y 594.787,Z 411.217,A -85,B 0,C 180,E1 27393.348,E2 27393.348} C_VEL
LIN {X 0,Y 593.368,Z 408.275,A -85,B 0,C 180,E1 27393.073,E2 27393.073} C_VEL
LIN {X 0,Y 593.192,Z 407.328,A -85,B 0,C 180,E1 27393.008,E2 27393.008} C_VEL
LIN {X 0,Y 593.181,Z 407.304,A -85,B 0,C 180,E1 27389.708,E2 27389.708} C_VEL
LIN {X 0,Y 593.183,Z 407.309,A -85,B 0,C 180,E1 27386.532,E2 27386.532} C_VEL
LIN {X 0,Y 593.177,Z 407.339,A -85,B 0,C 180,E1 27383.336,E2 27383.336} C_VEL
LIN {X 0,Y 593.182,Z 407.298,A -85,B 0,C 180,E1 27380.216,E2 27380.216} C_VEL
LIN {X 0,Y 593.176,Z 407.342,A -85,B 0,C 180,E1 27377.056,E2 27377.056} C_VEL
LIN {X 0,Y 593.183,Z 407.304,A -85,B 0,C 180,E1 27373.846,E2 27373.846} C_VEL
LIN {X 0,Y 593.174,Z 407.325,A -85,B 0,C 180,E1 27370.655,E2 27370.655} C_VEL
LIN {X 0,Y 593.196,Z 407.315,A -85,B 0,C 180,E1 27367.36,E2 27367.36} C_VEL
LIN {X 0,Y 593.183,Z 407.308,A -85,B 0,C 180,E1 27364.06,E2 27364.06} C_VEL
LIN {X 0,Y 593.179,Z 407.332,A -85,B 0,C 180,E1 27360.773,E2 27360.773} C_VEL
LIN {X 0,Y 593.188,Z 407.298,A -85,B 0,C 180,E1 27357.585,E2 27357.585} C_VEL
LIN {X 0,Y 593.167,Z 407.336,A -85,B 0,C 180,E1 27354.292,E2 27354.292} C_VEL
LIN {X 0,Y 593.188,Z 407.293,A -85,B 0,C 180,E1 27351.176,E2 27351.176} C_VEL
LIN {X 0,Y 593.165,Z 407.341,A -85,B 0,C 180,E1 27347.935,E2 27347.935} C_VEL
LIN {X 0,Y 593.19,Z 407.297,A -85,B 0,C 180,E1 27344.754,E2 27344.754} C_VEL
LIN {X 0,Y 593.165,Z 407.335,A -85,B 0,C 180,E1 27341.626,E2 27341.626} C_VEL
LIN {X 0,Y 593.199,Z 407.317,A -85,B 0,C 180,E1 27338.337,E2 27338.337} C_VEL
LIN {X 0,Y 593.168,Z 407.305,A -85,B 0,C 180,E1 27335.182,E2 27335.182} C_VEL
LIN {X 0,Y 593.177,Z 407.332,A -85,B 0,C 180,E1 27331.837,E2 27331.837} C_VEL
LIN {X 0,Y 593.189,Z 407.392,A -85,B 0,C 180,E1 27328.812,E2 27328.812} C_VEL
LIN {X 0,Y 594.477,Z 410.787,A -85,B 0,C 180,E1 27328.234,E2 27328.234} C_VEL
LIN {X 0,Y 595.733,Z 412.519,A -85,B 0,C 180,E1 27327.855,E2 27327.855} C_VEL
LIN {X 0,Y 597.577,Z 416.333,A -85,B 0,C 180,E1 27327.171,E2 27327.171} C_VEL
LIN {X 0,Y 601.19,Z 423.474,A -85,B 0,C 180,E1 27325.91,E2 27325.91} C_VEL
LIN {X 0,Y 608.409,Z 433.219,A -85,B 0,C 180,E1 27324.713,E2 27324.713} C_VEL
LIN {X 0,Y 618.495,Z 447.1,A -85,B 0,C 180,E1 27323.16,E2 27323.16} C_VEL
LIN {X 0,Y 630.438,Z 464.311,A -85,B 0,C 180,E1 27321.438,E2 27321.438} C_VEL
LIN {X 0,Y 640.302,Z 479.356,A -85,B 0,C 180,E1 27320.095,E2 27320.095} C_VEL
LIN {X 0,Y 634.963,Z 688.415,A -85,B 0,C 180,E1 27317.161,E2 27317.161} C_VEL
LIN {X 0,Y 629.782,Z 901.612,A -85,B 0,C 180,E1 27314.228,E2 27314.228} C_VEL
LIN {X 0,Y 628.727,Z 923.469,A -85,B 0,C 180,E1 27313.85,E2 27313.85} C_VEL
LIN {X 0,Y 627.287,Z 946.411,A -85,B 0,C 180,E1 27313.334,E2 27313.334} C_VEL
LIN {X 0,Y 625.098,Z 974.358,A -85,B 0,C 180,E1 27312.52,E2 27312.52} C_VEL
LIN {X 0,Y 622.971,Z 996.921,A -85,B 0,C 180,E1 27311.707,E2 27311.707} C_VEL
LIN {X 0,Y 620.858,Z 1017.51,A -85,B 0,C 180,E1 27310.836,E2 27310.836} C_VEL
LIN {X 0,Y 618.713,Z 1036.621,A -85,B 0,C 180,E1 27309.913,E2 27309.913} C_VEL
LIN {X 0,Y 616.348,Z 1056.284,A -85,B 0,C 180,E1 27308.839,E2 27308.839} C_VEL
LIN {X 0,Y 613.404,Z 1079.645,A -85,B 0,C 180,E1 27307.39,E2 27307.39} C_VEL
LIN {X 0,Y 610.276,Z 1102.515,A -85,B 0,C 180,E1 27305.742,E2 27305.742} C_VEL
LIN {X 0,Y 607.845,Z 1120.397,A -85,B 0,C 180,E1 27304.294,E2 27304.294} C_VEL
LIN {X 0,Y 605.439,Z 1138.232,A -85,B 0,C 180,E1 27302.69,E2 27302.69} C_VEL
LIN {X 0,Y 602.539,Z 1160.101,A -85,B 0,C 180,E1 27300.465,E2 27300.465} C_VEL
LIN {X 0,Y 600.36,Z 1176.65,A -85,B 0,C 180,E1 27298.558,E2 27298.558} C_VEL
LIN {X 0,Y 598.492,Z 1191.898,A -85,B 0,C 180,E1 27296.602,E2 27296.602} C_VEL
LIN {X 0,Y 596.566,Z 1208.879,A -85,B 0,C 180,E1 27294.143,E2 27294.143} C_VEL
LIN {X 0,Y 595.188,Z 1222.406,A -85,B 0,C 180,E1 27291.901,E2 27291.901} C_VEL
LIN {X 0,Y 594.183,Z 1233.794,A -85,B 0,C 180,E1 27289.773,E2 27289.773} C_VEL
LIN {X 0,Y 593.222,Z 1246.181,A -85,B 0,C 180,E1 27287.119,E2 27287.119} C_VEL
LIN {X 0,Y 592.673,Z 1255.436,A -85,B 0,C 180,E1 27284.762,E2 27284.762} C_VEL
LIN {X 0,Y 592.312,Z 1262.736,A -85,B 0,C 180,E1 27282.582,E2 27282.582} C_VEL
LIN {X 0,Y 592.12,Z 1268.554,A -85,B 0,C 180,E1 27280.512,E2 27280.512} C_VEL
LIN {X 0,Y 591.965,Z 1274.143,A -85,B 0,C 180,E1 27278.063,E2 27278.063} C_VEL
LIN {X 0,Y 591.922,Z 1278.422,A -85,B 0,C 180,E1 27275.432,E2 27275.432} C_VEL
LIN {X 0,Y 591.91,Z 1280.741,A -85,B 0,C 180,E1 27273.103,E2 27273.103} C_VEL
LIN {X 0,Y 591.879,Z 1281.758,A -85,B 0,C 180,E1 27271.069,E2 27271.069} C_VEL
LIN {X 0,Y 591.867,Z 1281.806,A -85,B 0,C 180,E1 27269.133,E2 27269.133} C_VEL
LIN {X 0,Y 591.91,Z 1280.951,A -85,B 0,C 180,E1 27267.197,E2 27267.197} C_VEL
LIN {X 0,Y 591.92,Z 1279.006,A -85,B 0,C 180,E1 27265.063,E2 27265.063} C_VEL
LIN {X 0,Y 591.952,Z 1275.431,A -85,B 0,C 180,E1 27262.629,E2 27262.629} C_VEL
LIN {X 0,Y 592.067,Z 1269.849,A -85,B 0,C 180,E1 27259.988,E2 27259.988} C_VEL
LIN {X 0,Y 592.267,Z 1263.672,A -85,B 0,C 180,E1 27257.724,E2 27257.724} C_VEL
LIN {X 0,Y 592.59,Z 1256.529,A -85,B 0,C 180,E1 27255.544,E2 27255.544} C_VEL
LIN {X 0,Y 593.069,Z 1248.515,A -85,B 0,C 180,E1 27253.451,E2 27253.451} C_VEL
LIN {X 0,Y 593.836,Z 1237.856,A -85,B 0,C 180,E1 27251.042,E2 27251.042} C_VEL
LIN {X 0,Y 594.96,Z 1224.756,A -85,B 0,C 180,E1 27248.514,E2 27248.514} C_VEL
LIN {X 0,Y 596.219,Z 1212.136,A -85,B 0,C 180,E1 27246.377,E2 27246.377} C_VEL
LIN {X 0,Y 597.804,Z 1197.906,A -85,B 0,C 180,E1 27244.229,E2 27244.229} C_VEL
LIN {X 0,Y 599.966,Z 1179.897,A -85,B 0,C 180,E1 27241.839,E2 27241.839} C_VEL
LIN {X 0,Y 602.059,Z 1163.427,A -85,B 0,C 180,E1 27239.904,E2 27239.904} C_VEL
LIN {X 0,Y 604.291,Z 1146.811,A -85,B 0,C 180,E1 27238.148,E2 27238.148} C_VEL
LIN {X 0,Y 607.349,Z 1124.34,A -85,B 0,C 180,E1 27236.043,E2 27236.043} C_VEL
LIN {X 0,Y 609.897,Z 1105.3,A -85,B 0,C 180,E1 27234.474,E2 27234.474} C_VEL
LIN {X 0,Y 612.432,Z 1086.394,A -85,B 0,C 180,E1 27233.08,E2 27233.08} C_VEL
LIN {X 0,Y 615.445,Z 1063.597,A -85,B 0,C 180,E1 27231.587,E2 27231.587} C_VEL
LIN {X 0,Y 618.343,Z 1039.825,A -85,B 0,C 180,E1 27230.251,E2 27230.251} C_VEL
LIN {X 0,Y 620.583,Z 1019.981,A -85,B 0,C 180,E1 27229.275,E2 27229.275} C_VEL
LIN {X 0,Y 622.685,Z 999.726,A -85,B 0,C 180,E1 27228.404,E2 27228.404} C_VEL
LIN {X 0,Y 624.645,Z 979.067,A -85,B 0,C 180,E1 27227.639,E2 27227.639} C_VEL
LIN {X 0,Y 626.489,Z 957.042,A -85,B 0,C 180,E1 27226.952,E2 27226.952} C_VEL
LIN {X 0,Y 628.43,Z 929.309,A -85,B 0,C 180,E1 27226.265,E2 27226.265} C_VEL
LIN {X 0,Y 629.683,Z 904.175,A -85,B 0,C 180,E1 27225.81,E2 27225.81} C_VEL
LIN {X 0,Y 632.902,Z 773.755,A -85,B 0,C 180,E1 27224.015,E2 27224.015} C_VEL
LIN {X 0,Y 638.224,Z 558.808,A -85,B 0,C 180,E1 27221.029,E2 27221.029} C_VEL
LIN {X 0,Y 640.214,Z 479.059,A -85,B 0,C 180,E1 27219.89,E2 27219.89} C_VEL
LIN {X 0,Y 624.848,Z 456.022,A -85,B 0,C 180,E1 27217.769,E2 27217.769} C_VEL
LIN {X 0,Y 613.291,Z 439.919,A -85,B 0,C 180,E1 27216.055,E2 27216.055} C_VEL
LIN {X 0,Y 605.839,Z 429.791,A -85,B 0,C 180,E1 27214.881,E2 27214.881} C_VEL
LIN {X 0,Y 601.151,Z 423.434,A -85,B 0,C 180,E1 27214.086,E2 27214.086} C_VEL
LIN {X 0,Y 599.794,Z 420.616,A -85,B 0,C 180,E1 27213.605,E2 27213.605} C_VEL
LIN {X 0,Y 597.542,Z 416.327,A -85,B 0,C 180,E1 27212.831,E2 27212.831} C_VEL
LIN {X 0,Y 595.709,Z 412.487,A -85,B 0,C 180,E1 27212.146,E2 27212.146} C_VEL
LIN {X 0,Y 593.427,Z 408.639,A -85,B 0,C 180,E1 27211.376,E2 27211.376} C_VEL
LIN {X 0,Y 593.137,Z 407.328,A -85,B 0,C 180,E1 27211.167,E2 27211.167} C_VEL
LIN {X 0,Y 593.15,Z 407.329,A -85,B 0,C 180,E1 27208.274,E2 27208.274} C_VEL
LIN {X 0,Y 593.127,Z 407.307,A -85,B 0,C 180,E1 27205.033,E2 27205.033} C_VEL
LIN {X 0,Y 593.134,Z 407.343,A -85,B 0,C 180,E1 27202.186,E2 27202.186} C_VEL
LIN {X 0,Y 593.119,Z 407.324,A -85,B 0,C 180,E1 27198.886,E2 27198.886} C_VEL
LIN {X 0,Y 593.119,Z 407.321,A -85,B 0,C 180,E1 27196.05,E2 27196.05} C_VEL
LIN {X 0,Y 593.112,Z 407.344,A -85,B 0,C 180,E1 27192.759,E2 27192.759} C_VEL
LIN {X 0,Y 593.107,Z 407.312,A -85,B 0,C 180,E1 27189.902,E2 27189.902} C_VEL
LIN {X 0,Y 593.104,Z 407.351,A -85,B 0,C 180,E1 27186.583,E2 27186.583} C_VEL
LIN {X 0,Y 593.109,Z 407.308,A -85,B 0,C 180,E1 27183.728,E2 27183.728} C_VEL
LIN {X 0,Y 593.113,Z 407.349,A -85,B 0,C 180,E1 27180.386,E2 27180.386} C_VEL
LIN {X 0,Y 593.117,Z 407.306,A -85,B 0,C 180,E1 27177.584,E2 27177.584} C_VEL
LIN {X 0,Y 593.127,Z 407.348,A -85,B 0,C 180,E1 27174.292,E2 27174.292} C_VEL
LIN {X 0,Y 593.12,Z 407.307,A -85,B 0,C 180,E1 27171.566,E2 27171.566} C_VEL
LIN {X 0,Y 593.153,Z 407.346,A -85,B 0,C 180,E1 27168.313,E2 27168.313} C_VEL
LIN {X 0,Y 593.128,Z 407.305,A -85,B 0,C 180,E1 27165.452,E2 27165.452} C_VEL
LIN {X 0,Y 593.171,Z 407.343,A -85,B 0,C 180,E1 27162.226,E2 27162.226} C_VEL
LIN {X 0,Y 593.137,Z 407.302,A -85,B 0,C 180,E1 27159.267,E2 27159.267} C_VEL
LIN {X 0,Y 593.173,Z 407.333,A -85,B 0,C 180,E1 27156.031,E2 27156.031} C_VEL
LIN {X 0,Y 593.161,Z 407.325,A -85,B 0,C 180,E1 27152.926,E2 27152.926} C_VEL
LIN {X 0,Y 593.157,Z 407.303,A -85,B 0,C 180,E1 27149.621,E2 27149.621} C_VEL
LIN {X 0,Y 593.19,Z 407.535,A -85,B 0,C 180,E1 27146.871,E2 27146.871} C_VEL
LIN {X 0,Y 594.264,Z 410.464,A -85,B 0,C 180,E1 27146.648,E2 27146.648} C_VEL
LIN {X 0,Y 596.878,Z 413.093,A -85,B 0,C 180,E1 27146.209,E2 27146.209} C_VEL
LIN {X 0,Y 597.899,Z 413.945,A -85,B 0,C 180,E1 27146.043,E2 27146.043} C_VEL
LIN {X 0,Y 600.302,Z 417.74,A -85,B 0,C 180,E1 27145.622,E2 27145.622} C_VEL
LIN {X 0,Y 602.74,Z 420.112,A -85,B 0,C 180,E1 27145.232,E2 27145.232} C_VEL
LIN {X 0,Y 605.883,Z 424.295,A -85,B 0,C 180,E1 27144.717,E2 27144.717} C_VEL
LIN {X 0,Y 607.555,Z 426.289,A -85,B 0,C 180,E1 27144.453,E2 27144.453} C_VEL
LIN {X 0,Y 613.122,Z 433.421,A -85,B 0,C 180,E1 27143.586,E2 27143.586} C_VEL
LIN {X 0,Y 617.215,Z 438.629,A -85,B 0,C 180,E1 27142.97,E2 27142.97} C_VEL
LIN {X 0,Y 627.894,Z 452.596,A -85,B 0,C 180,E1 27141.432,E2 27141.432} C_VEL
LIN {X 0,Y 640.041,Z 469.423,A -85,B 0,C 180,E1 27139.786,E2 27139.786} C_VEL
LIN {X 0,Y 635.541,Z 641.388,A -85,B 0,C 180,E1 27137.366,E2 27137.366} C_VEL
LIN {X 0,Y 634.667,Z 649.091,A -85,B 0,C 180,E1 27137.325,E2 27137.325} C_VEL
LIN {X 0,Y 629.922,Z 669.75,A -85,B 0,C 180,E1 27137.456,E2 27137.456} C_VEL
LIN {X 0,Y 629.23,Z 676.359,A -85,B 0,C 180,E1 27137.416,E2 27137.416} C_VEL
LIN {X 0,Y 624.011,Z 874.274,A -85,B 0,C 180,E1 27134.663,E2 27134.663} C_VEL
LIN {X 0,Y 622.773,Z 897.969,A -85,B 0,C 180,E1 27134.234,E2 27134.234} C_VEL
LIN {X 0,Y 620.709,Z 926.394,A -85,B 0,C 180,E1 27133.537,E2 27133.537} C_VEL
LIN {X 0,Y 618.795,Z 948.138,A -85,B 0,C 180,E1 27132.857,E2 27132.857} C_VEL
LIN {X 0,Y 616.712,Z 968.8,A -85,B 0,C 180,E1 27132.09,E2 27132.09} C_VEL
LIN {X 0,Y 614.501,Z 989.157,A -85,B 0,C 180,E1 27131.215,E2 27131.215} C_VEL
LIN {X 0,Y 612.133,Z 1009.084,A -85,B 0,C 180,E1 27130.234,E2 27130.234} C_VEL
LIN {X 0,Y 609.099,Z 1032.908,A -85,B 0,C 180,E1 27128.894,E2 27128.894} C_VEL
LIN {X 0,Y 605.886,Z 1055.835,A -85,B 0,C 180,E1 27127.387,E2 27127.387} C_VEL
LIN {X 0,Y 603.205,Z 1074.719,A -85,B 0,C 180,E1 27125.987,E2 27125.987} C_VEL
LIN {X 0,Y 600.49,Z 1093.68,A -85,B 0,C 180,E1 27124.416,E2 27124.416} C_VEL
LIN {X 0,Y 597.237,Z 1116.408,A -85,B 0,C 180,E1 27122.273,E2 27122.273} C_VEL
LIN {X 0,Y 594.876,Z 1133.052,A -85,B 0,C 180,E1 27120.498,E2 27120.498} C_VEL
LIN {X 0,Y 592.776,Z 1148.266,A -85,B 0,C 180,E1 27118.701,E2 27118.701} C_VEL
LIN {X 0,Y 590.569,Z 1165.661,A -85,B 0,C 180,E1 27116.408,E2 27116.408} C_VEL
LIN {X 0,Y 588.652,Z 1181.231,A -85,B 0,C 180,E1 27114.052,E2 27114.052} C_VEL
LIN {X 0,Y 587.356,Z 1193.362,A -85,B 0,C 180,E1 27111.988,E2 27111.988} C_VEL
LIN {X 0,Y 586.166,Z 1206.194,A -85,B 0,C 180,E1 27109.526,E2 27109.526} C_VEL
LIN {X 0,Y 585.199,Z 1217.928,A -85,B 0,C 180,E1 27106.88,E2 27106.88} C_VEL
LIN {X 0,Y 584.678,Z 1226.371,A -85,B 0,C 180,E1 27104.656,E2 27104.656} C_VEL
LIN {X 0,Y 584.305,Z 1233.536,A -85,B 0,C 180,E1 27102.446,E2 27102.446} C_VEL
LIN {X 0,Y 584.069,Z 1240.242,A -85,B 0,C 180,E1 27099.952,E2 27099.952} C_VEL
LIN {X 0,Y 583.951,Z 1245.519,A -85,B 0,C 180,E1 27097.373,E2 27097.373} C_VEL
LIN {X 0,Y 583.921,Z 1248.951,A -85,B 0,C 180,E1 27095.005,E2 27095.005} C_VEL
LIN {X 0,Y 583.91,Z 1250.919,A -85,B 0,C 180,E1 27092.842,E2 27092.842} C_VEL
LIN {X 0,Y 583.868,Z 1251.818,A -85,B 0,C 180,E1 27090.78,E2 27090.78} C_VEL
LIN {X 0,Y 583.89,Z 1251.723,A -85,B 0,C 180,E1 27088.72,E2 27088.72} C_VEL
LIN {X 0,Y 583.912,Z 1250.499,A -85,B 0,C 180,E1 27086.461,E2 27086.461} C_VEL
LIN {X 0,Y 583.944,Z 1247.547,A -85,B 0,C 180,E1 27083.803,E2 27083.803} C_VEL
LIN {X 0,Y 584.011,Z 1243.011,A -85,B 0,C 180,E1 27081.231,E2 27081.231} C_VEL
LIN {X 0,Y 584.146,Z 1237.651,A -85,B 0,C 180,E1 27078.943,E2 27078.943} C_VEL
LIN {X 0,Y 584.425,Z 1231.349,A -85,B 0,C 180,E1 27076.743,E2 27076.743} C_VEL
LIN {X 0,Y 584.947,Z 1221.896,A -85,B 0,C 180,E1 27074.022,E2 27074.022} C_VEL
LIN {X 0,Y 585.632,Z 1212.13,A -85,B 0,C 180,E1 27071.678,E2 27071.678} C_VEL
LIN {X 0,Y 586.528,Z 1201.956,A -85,B 0,C 180,E1 27069.541,E2 27069.541} C_VEL
LIN {X 0,Y 587.816,Z 1189.183,A -85,B 0,C 180,E1 27067.177,E2 27067.177} C_VEL
LIN {X 0,Y 589.552,Z 1173.7,A -85,B 0,C 180,E1 27064.686,E2 27064.686} C_VEL
LIN {X 0,Y 591.234,Z 1159.903,A -85,B 0,C 180,E1 27062.718,E2 27062.718} C_VEL
LIN {X 0,Y 593.226,Z 1145.112,A -85,B 0,C 180,E1 27060.821,E2 27060.821} C_VEL
LIN {X 0,Y 595.866,Z 1126.243,A -85,B 0,C 180,E1 27058.652,E2 27058.652} C_VEL
LIN {X 0,Y 598.563,Z 1107.002,A -85,B 0,C 180,E1 27056.715,E2 27056.715} C_VEL
LIN {X 0,Y 601.068,Z 1089.651,A -85,B 0,C 180,E1 27055.148,E2 27055.148} C_VEL
LIN {X 0,Y 603.769,Z 1071.02,A -85,B 0,C 180,E1 27053.636,E2 27053.636} C_VEL
LIN {X 0,Y 607.164,Z 1047.096,A -85,B 0,C 180,E1 27051.923,E2 27051.923} C_VEL
LIN {X 0,Y 609.951,Z 1026.137,A -85,B 0,C 180,E1 27050.621,E2 27050.621} C_VEL
LIN {X 0,Y 612.468,Z 1006.304,A -85,B 0,C 180,E1 27049.533,E2 27049.533} C_VEL
LIN {X 0,Y 614.729,Z 987.194,A -85,B 0,C 180,E1 27048.606,E2 27048.606} C_VEL
LIN {X 0,Y 616.949,Z 966.566,A -85,B 0,C 180,E1 27047.73,E2 27047.73} C_VEL
LIN {X 0,Y 619.429,Z 941.853,A -85,B 0,C 180,E1 27046.838,E2 27046.838} C_VEL
LIN {X 0,Y 621.571,Z 915.2,A -85,B 0,C 180,E1 27046.075,E2 27046.075} C_VEL
LIN {X 0,Y 623.01,Z 893.494,A -85,B 0,C 180,E1 27045.586,E2 27045.586} C_VEL
LIN {X 0,Y 624.106,Z 871.836,A -85,B 0,C 180,E1 27045.21,E2 27045.21} C_VEL
LIN {X 0,Y 629.676,Z 659.292,A -85,B 0,C 180,E1 27042.255,E2 27042.255} C_VEL
LIN {X 0,Y 634.773,Z 473.491,A -85,B 0,C 180,E1 27039.624,E2 27039.624} C_VEL
LIN {X 0,Y 622.189,Z 456.117,A -85,B 0,C 180,E1 27037.872,E2 27037.872} C_VEL
LIN {X 0,Y 611.398,Z 441.917,A -85,B 0,C 180,E1 27036.265,E2 27036.265} C_VEL
LIN {X 0,Y 606.368,Z 435.659,A -85,B 0,C 180,E1 27035.482,E2 27035.482} C_VEL
LIN {X 0,Y 602.94,Z 431.234,A -85,B 0,C 180,E1 27034.928,E2 27034.928} C_VEL
LIN {X 0,Y 598.683,Z 425.881,A -85,B 0,C 180,E1 27034.224,E2 27034.224} C_VEL
LIN {X 0,Y 595.468,Z 422.001,A -85,B 0,C 180,E1 27033.68,E2 27033.68} C_VEL
LIN {X 0,Y 594.391,Z 420.43,A -85,B 0,C 180,E1 27033.488,E2 27033.488} C_VEL
LIN {X 0,Y 591.309,Z 417.282,A -85,B 0,C 180,E1 27032.962,E2 27032.962} C_VEL
LIN {X 0,Y 589.833,Z 414.604,A -85,B 0,C 180,E1 27032.679,E2 27032.679} C_VEL
LIN {X 0,Y 586.996,Z 412.4,A -85,B 0,C 180,E1 27032.191,E2 27032.191} C_VEL
LIN {X 0,Y 585.462,Z 409.404,A -85,B 0,C 180,E1 27031.881,E2 27031.881} C_VEL
LIN {X 0,Y 585.247,Z 408.313,A -85,B 0,C 180,E1 27031.813,E2 27031.813} C_VEL
LIN {X 0,Y 585.245,Z 408.318,A -85,B 0,C 180,E1 27028.575,E2 27028.575} C_VEL
LIN {X 0,Y 585.235,Z 408.286,A -85,B 0,C 180,E1 27025.333,E2 27025.333} C_VEL
LIN {X 0,Y 585.247,Z 408.32,A -85,B 0,C 180,E1 27022.177,E2 27022.177} C_VEL
LIN {X 0,Y 585.236,Z 408.307,A -85,B 0,C 180,E1 27018.943,E2 27018.943} C_VEL
LIN {X 0,Y 585.253,Z 408.29,A -85,B 0,C 180,E1 27015.661,E2 27015.661} C_VEL
LIN {X 0,Y 585.253,Z 408.325,A -85,B 0,C 180,E1 27012.331,E2 27012.331} C_VEL
LIN {X 0,Y 585.236,Z 408.28,A -85,B 0,C 180,E1 27009.044,E2 27009.044} C_VEL
LIN {X 0,Y 585.256,Z 408.332,A -85,B 0,C 180,E1 27005.884,E2 27005.884} C_VEL
LIN {X 0,Y 585.227,Z 408.279,A -85,B 0,C 180,E1 27002.644,E2 27002.644} C_VEL
LIN {X 0,Y 585.252,Z 408.328,A -85,B 0,C 180,E1 26999.511,E2 26999.511} C_VEL
LIN {X 0,Y 585.223,Z 408.279,A -85,B 0,C 180,E1 26996.277,E2 26996.277} C_VEL
LIN {X 0,Y 585.255,Z 408.321,A -85,B 0,C 180,E1 26993.033,E2 26993.033} C_VEL
LIN {X 0,Y 585.231,Z 408.29,A -85,B 0,C 180,E1 26989.765,E2 26989.765} C_VEL
LIN {X 0,Y 585.247,Z 408.305,A -85,B 0,C 180,E1 26986.447,E2 26986.447} C_VEL
LIN {X 0,Y 585.25,Z 408.316,A -85,B 0,C 180,E1 26983.218,E2 26983.218} C_VEL
LIN {X 0,Y 585.224,Z 408.287,A -85,B 0,C 180,E1 26979.914,E2 26979.914} C_VEL
LIN {X 0,Y 585.259,Z 408.324,A -85,B 0,C 180,E1 26976.756,E2 26976.756} C_VEL
LIN {X 0,Y 585.222,Z 408.307,A -85,B 0,C 180,E1 26973.517,E2 26973.517} C_VEL
LIN {X 0,Y 585.256,Z 408.287,A -85,B 0,C 180,E1 26970.413,E2 26970.413} C_VEL
LIN {X 0,Y 585.271,Z 408.453,A -85,B 0,C 180,E1 26969.932,E2 26969.932} C_VEL
LIN {X 0,Y 586.48,Z 411.72,A -85,B 0,C 180,E1 26969.352,E2 26969.352} C_VEL
LIN {X 0,Y 587.963,Z 413.875,A -85,B 0,C 180,E1 26968.87,E2 26968.87} C_VEL
LIN {X 0,Y 589.796,Z 417.473,A -85,B 0,C 180,E1 26968.18,E2 26968.18} C_VEL
LIN {X 0,Y 593.157,Z 423.714,A -85,B 0,C 180,E1 26967.039,E2 26967.039} C_VEL
LIN {X 0,Y 605.021,Z 439.607,A -85,B 0,C 180,E1 26965.036,E2 26965.036} C_VEL
LIN {X 0,Y 615.079,Z 453.593,A -85,B 0,C 180,E1 26963.46,E2 26963.46} C_VEL
LIN {X 0,Y 626.703,Z 470.494,A -85,B 0,C 180,E1 26961.753,E2 26961.753} C_VEL
LIN {X 0,Y 635.041,Z 483.229,A -85,B 0,C 180,E1 26960.594,E2 26960.594} C_VEL
LIN {X 0,Y 629.349,Z 694.468,A -85,B 0,C 180,E1 26957.611,E2 26957.611} C_VEL
LIN {X 0,Y 623.998,Z 902.315,A -85,B 0,C 180,E1 26954.729,E2 26954.729} C_VEL
LIN {X 0,Y 622.85,Z 924.671,A -85,B 0,C 180,E1 26954.336,E2 26954.336} C_VEL
LIN {X 0,Y 621.074,Z 951.406,A -85,B 0,C 180,E1 26953.714,E2 26953.714} C_VEL
LIN {X 0,Y 618.833,Z 977.189,A -85,B 0,C 180,E1 26952.928,E2 26952.928} C_VEL
LIN {X 0,Y 616.773,Z 998.204,A -85,B 0,C 180,E1 26952.159,E2 26952.159} C_VEL
LIN {X 0,Y 614.561,Z 1018.637,A -85,B 0,C 180,E1 26951.283,E2 26951.283} C_VEL
LIN {X 0,Y 612.187,Z 1038.628,A -85,B 0,C 180,E1 26950.303,E2 26950.303} C_VEL
LIN {X 0,Y 609.14,Z 1062.633,A -85,B 0,C 180,E1 26948.956,E2 26948.956} C_VEL
LIN {X 0,Y 605.965,Z 1085.33,A -85,B 0,C 180,E1 26947.468,E2 26947.468} C_VEL
LIN {X 0,Y 603.237,Z 1104.515,A -85,B 0,C 180,E1 26946.048,E2 26946.048} C_VEL
LIN {X 0,Y 600.527,Z 1123.437,A -85,B 0,C 180,E1 26944.482,E2 26944.482} C_VEL
LIN {X 0,Y 597.273,Z 1146.168,A -85,B 0,C 180,E1 26942.343,E2 26942.343} C_VEL
LIN {X 0,Y 594.903,Z 1162.877,A -85,B 0,C 180,E1 26940.562,E2 26940.562} C_VEL
LIN {X 0,Y 592.713,Z 1178.721,A -85,B 0,C 180,E1 26938.69,E2 26938.69} C_VEL
LIN {X 0,Y 590.468,Z 1196.423,A -85,B 0,C 180,E1 26936.341,E2 26936.341} C_VEL
LIN {X 0,Y 588.628,Z 1211.439,A -85,B 0,C 180,E1 26934.063,E2 26934.063} C_VEL
LIN {X 0,Y 587.335,Z 1223.551,A -85,B 0,C 180,E1 26931.999,E2 26931.999} C_VEL
LIN {X 0,Y 586.111,Z 1236.875,A -85,B 0,C 180,E1 26929.434,E2 26929.434} C_VEL
LIN {X 0,Y 585.191,Z 1248.07,A -85,B 0,C 180,E1 26926.89,E2 26926.89} C_VEL
LIN {X 0,Y 584.695,Z 1256.144,A -85,B 0,C 180,E1 26924.766,E2 26924.766} C_VEL
LIN {X 0,Y 584.32,Z 1263.342,A -85,B 0,C 180,E1 26922.556,E2 26922.556} C_VEL
LIN {X 0,Y 584.106,Z 1269.571,A -85,B 0,C 180,E1 26920.259,E2 26920.259} C_VEL
LIN {X 0,Y 583.949,Z 1275.244,A -85,B 0,C 180,E1 26917.58,E2 26917.58} C_VEL
LIN {X 0,Y 583.921,Z 1278.88,A -85,B 0,C 180,E1 26915.113,E2 26915.113} C_VEL
LIN {X 0,Y 583.91,Z 1280.876,A -85,B 0,C 180,E1 26912.949,E2 26912.949} C_VEL
LIN {X 0,Y 583.874,Z 1281.781,A -85,B 0,C 180,E1 26910.986,E2 26910.986} C_VEL
LIN {X 0,Y 583.873,Z 1281.783,A -85,B 0,C 180,E1 26909.023,E2 26909.023} C_VEL
LIN {X 0,Y 583.91,Z 1280.882,A -85,B 0,C 180,E1 26907.06,E2 26907.06} C_VEL
LIN {X 0,Y 583.922,Z 1278.889,A -85,B 0,C 180,E1 26904.896,E2 26904.896} C_VEL
LIN {X 0,Y 583.948,Z 1275.259,A -85,B 0,C 180,E1 26902.429,E2 26902.429} C_VEL
LIN {X 0,Y 584.106,Z 1269.594,A -85,B 0,C 180,E1 26899.75,E2 26899.75} C_VEL
LIN {X 0,Y 584.317,Z 1263.368,A -85,B 0,C 180,E1 26897.453,E2 26897.453} C_VEL
LIN {X 0,Y 584.693,Z 1256.175,A -85,B 0,C 180,E1 26895.243,E2 26895.243} C_VEL
LIN {X 0,Y 585.217,Z 1247.698,A -85,B 0,C 180,E1 26893.018,E2 26893.018} C_VEL
LIN {X 0,Y 586.216,Z 1235.601,A -85,B 0,C 180,E1 26890.311,E2 26890.311} C_VEL
LIN {X 0,Y 587.328,Z 1223.607,A -85,B 0,C 180,E1 26888.011,E2 26888.011} C_VEL
LIN {X 0,Y 588.62,Z 1211.499,A -85,B 0,C 180,E1 26885.947,E2 26885.947} C_VEL
LIN {X 0,Y 590.555,Z 1195.776,A -85,B 0,C 180,E1 26883.564,E2 26883.564} C_VEL
LIN {X 0,Y 592.752,Z 1178.416,A -85,B 0,C 180,E1 26881.272,E2 26881.272} C_VEL
LIN {X 0,Y 594.959,Z 1162.499,A -85,B 0,C 180,E1 26879.395,E2 26879.395} C_VEL
LIN {X 0,Y 597.639,Z 1143.766,A -85,B 0,C 180,E1 26877.41,E2 26877.41} C_VEL
LIN {X 0,Y 600.677,Z 1122.328,A -85,B 0,C 180,E1 26875.422,E2 26875.422} C_VEL
LIN {X 0,Y 603.316,Z 1103.962,A -85,B 0,C 180,E1 26873.909,E2 26873.909} C_VEL
LIN {X 0,Y 606.023,Z 1084.921,A -85,B 0,C 180,E1 26872.504,E2 26872.504} C_VEL
LIN {X 0,Y 609.461,Z 1060.121,A -85,B 0,C 180,E1 26870.897,E2 26870.897} C_VEL
LIN {X 0,Y 612.167,Z 1038.817,A -85,B 0,C 180,E1 26869.707,E2 26869.707} C_VEL
LIN {X 0,Y 614.494,Z 1019.219,A -85,B 0,C 180,E1 26868.743,E2 26868.743} C_VEL
LIN {X 0,Y 616.612,Z 999.723,A -85,B 0,C 180,E1 26867.901,E2 26867.901} C_VEL
LIN {X 0,Y 618.587,Z 979.697,A -85,B 0,C 180,E1 26867.157,E2 26867.157} C_VEL
LIN {X 0,Y 620.463,Z 958.167,A -85,B 0,C 180,E1 26866.479,E2 26866.479} C_VEL
LIN {X 0,Y 622.469,Z 931.706,A -85,B 0,C 180,E1 26865.806,E2 26865.806} C_VEL
LIN {X 0,Y 623.909,Z 904.555,A -85,B 0,C 180,E1 26865.305,E2 26865.305} C_VEL
LIN {X 0,Y 626.398,Z 810.816,A -85,B 0,C 180,E1 26864.001,E2 26864.001} C_VEL
LIN {X 0,Y 632.008,Z 593.611,A -85,B 0,C 180,E1 26860.974,E2 26860.974} C_VEL
LIN {X 0,Y 634.96,Z 482.935,A -85,B 0,C 180,E1 26859.392,E2 26859.392} C_VEL
LIN {X 0,Y 619.825,Z 460.444,A -85,B 0,C 180,E1 26857.254,E2 26857.254} C_VEL
LIN {X 0,Y 610.373,Z 447.005,A -85,B 0,C 180,E1 26855.82,E2 26855.82} C_VEL
LIN {X 0,Y 602.47,Z 436.205,A -85,B 0,C 180,E1 26854.554,E2 26854.554} C_VEL
LIN {X 0,Y 594.916,Z 426.284,A -85,B 0,C 180,E1 26853.282,E2 26853.282} C_VEL
LIN {X 0,Y 592.692,Z 422.813,A -85,B 0,C 180,E1 26852.846,E2 26852.846} C_VEL
LIN {X 0,Y 590.554,Z 419.033,A -85,B 0,C 180,E1 26852.117,E2 26852.117} C_VEL
LIN {X 0,Y 589.148,Z 416.572,A -85,B 0,C 180,E1 26851.63,E2 26851.63} C_VEL
LIN {X 0,Y 587.298,Z 412.8,A -85,B 0,C 180,E1 26850.914,E2 26850.914} C_VEL
LIN {X 0,Y 585.491,Z 409.593,A -85,B 0,C 180,E1 26850.252,E2 26850.252} C_VEL
LIN {X 0,Y 585.244,Z 408.288,A -85,B 0,C 180,E1 26850.039,E2 26850.039} C_VEL
LIN {X 0,Y 585.188,Z 408.325,A -85,B 0,C 180,E1 26846.901,E2 26846.901} C_VEL
LIN {X 0,Y 585.247,Z 408.309,A -85,B 0,C 180,E1 26843.779,E2 26843.779} C_VEL
LIN {X 0,Y 585.172,Z 408.296,A -85,B 0,C 180,E1 26840.714,E2 26840.714} C_VEL
LIN {X 0,Y 585.242,Z 408.333,A -85,B 0,C 180,E1 26837.596,E2 26837.596} C_VEL
LIN {X 0,Y 585.16,Z 408.294,A -85,B 0,C 180,E1 26834.548,E2 26834.548} C_VEL
LIN {X 0,Y 585.22,Z 408.331,A -85,B 0,C 180,E1 26831.531,E2 26831.531} C_VEL
LIN {X 0,Y 585.148,Z 408.3,A -85,B 0,C 180,E1 26828.352,E2 26828.352} C_VEL
LIN {X 0,Y 585.213,Z 408.327,A -85,B 0,C 180,E1 26825.392,E2 26825.392} C_VEL
LIN {X 0,Y 585.156,Z 408.3,A -85,B 0,C 180,E1 26822.252,E2 26822.252} C_VEL
LIN {X 0,Y 585.202,Z 408.331,A -85,B 0,C 180,E1 26819.413,E2 26819.413} C_VEL
LIN {X 0,Y 585.17,Z 408.298,A -85,B 0,C 180,E1 26816.158,E2 26816.158} C_VEL
LIN {X 0,Y 585.214,Z 408.327,A -85,B 0,C 180,E1 26813.229,E2 26813.229} C_VEL
LIN {X 0,Y 585.183,Z 408.297,A -85,B 0,C 180,E1 26810.062,E2 26810.062} C_VEL
LIN {X 0,Y 585.212,Z 408.325,A -85,B 0,C 180,E1 26807.166,E2 26807.166} C_VEL
LIN {X 0,Y 585.196,Z 408.303,A -85,B 0,C 180,E1 26803.931,E2 26803.931} C_VEL
LIN {X 0,Y 585.227,Z 408.307,A -85,B 0,C 180,E1 26800.954,E2 26800.954} C_VEL
LIN {X 0,Y 585.204,Z 408.323,A -85,B 0,C 180,E1 26797.709,E2 26797.709} C_VEL
LIN {X 0,Y 585.249,Z 408.287,A -85,B 0,C 180,E1 26794.607,E2 26794.607} C_VEL
LIN {X 0,Y 585.211,Z 408.326,A -85,B 0,C 180,E1 26791.413,E2 26791.413} C_VEL
LIN {X 0,Y 585.259,Z 408.305,A -85,B 0,C 180,E1 26788.286,E2 26788.286} C_VEL
LIN {X 0,Y 585.282,Z 408.492,A -85,B 0,C 180,E1 26788.067,E2 26788.067} C_VEL
LIN {X 0,Y 586.363,Z 411.517,A -85,B 0,C 180,E1 26787.828,E2 26787.828} C_VEL
LIN {X 0,Y 588.887,Z 414.113,A -85,B 0,C 180,E1 26787.378,E2 26787.378} C_VEL
LIN {X 0,Y 590.059,Z 414.976,A -85,B 0,C 180,E1 26787.18,E2 26787.18} C_VEL
LIN {X 0,Y 592.338,Z 418.61,A -85,B 0,C 180,E1 26786.757,E2 26786.757} C_VEL
LIN {X 0,Y 594.953,Z 421.14,A -85,B 0,C 180,E1 26786.316,E2 26786.316} C_VEL
LIN {X 0,Y 597.999,Z 425.277,A -85,B 0,C 180,E1 26785.79,E2 26785.79} C_VEL
LIN {X 0,Y 599.892,Z 427.345,A -85,B 0,C 180,E1 26785.479,E2 26785.479} C_VEL
LIN {X 0,Y 605.055,Z 433.996,A -85,B 0,C 180,E1 26784.633,E2 26784.633} C_VEL
LIN {X 0,Y 610.217,Z 440.493,A -85,B 0,C 180,E1 26783.822,E2 26783.822} C_VEL
LIN {X 0,Y 618,Z 450.574,A -85,B 0,C 180,E1 26782.646,E2 26782.646} C_VEL
LIN {X 0,Y 631.015,Z 468.102,A -85,B 0,C 180,E1 26780.798,E2 26780.798} C_VEL
LIN {X 0,Y 634.788,Z 473.904,A -85,B 0,C 180,E1 26780.277,E2 26780.277} C_VEL
LIN {X 0,Y 629.23,Z 676.359,A -85,B 0,C 180,E1 26777.416,E2 26777.416} C_VEL
LIN {X 0,Y 628.339,Z 684.064,A -85,B 0,C 180,E1 26777.377,E2 26777.377} C_VEL
LIN {X 0,Y 623.567,Z 704.715,A -85,B 0,C 180,E1 26777.512,E2 26777.512} C_VEL
LIN {X 0,Y 622.882,Z 711.323,A -85,B 0,C 180,E1 26777.471,E2 26777.471} C_VEL
LIN {X 0,Y 618.339,Z 874.686,A -85,B 0,C 180,E1 26775.183,E2 26775.183} C_VEL
LIN {X 0,Y 617.028,Z 898.75,A -85,B 0,C 180,E1 26774.744,E2 26774.744} C_VEL
LIN {X 0,Y 614.862,Z 927.106,A -85,B 0,C 180,E1 26774.04,E2 26774.04} C_VEL
LIN {X 0,Y 612.905,Z 948.421,A -85,B 0,C 180,E1 26773.37,E2 26773.37} C_VEL
LIN {X 0,Y 610.723,Z 969.076,A -85,B 0,C 180,E1 26772.6,E2 26772.6} C_VEL
LIN {X 0,Y 608.469,Z 988.645,A -85,B 0,C 180,E1 26771.75,E2 26771.75} C_VEL
LIN {X 0,Y 605.949,Z 1008.57,A -85,B 0,C 180,E1 26770.764,E2 26770.764} C_VEL
LIN {X 0,Y 602.808,Z 1032.161,A -85,B 0,C 180,E1 26769.433,E2 26769.433} C_VEL
LIN {X 0,Y 599.392,Z 1055.355,A -85,B 0,C 180,E1 26767.903,E2 26767.903} C_VEL
LIN {X 0,Y 596.583,Z 1074.124,A -85,B 0,C 180,E1 26766.504,E2 26766.504} C_VEL
LIN {X 0,Y 593.788,Z 1092.47,A -85,B 0,C 180,E1 26764.978,E2 26764.978} C_VEL
LIN {X 0,Y 590.565,Z 1113.879,A -85,B 0,C 180,E1 26762.972,E2 26762.972} C_VEL
LIN {X 0,Y 587.802,Z 1132.131,A -85,B 0,C 180,E1 26761.019,E2 26761.019} C_VEL
LIN {X 0,Y 585.584,Z 1147.229,A -85,B 0,C 180,E1 26759.225,E2 26759.225} C_VEL
LIN {X 0,Y 583.406,Z 1162.684,A -85,B 0,C 180,E1 26757.188,E2 26757.188} C_VEL
LIN {X 0,Y 581.187,Z 1179.963,A -85,B 0,C 180,E1 26754.597,E2 26754.597} C_VEL
LIN {X 0,Y 579.695,Z 1192.791,A -85,B 0,C 180,E1 26752.401,E2 26752.401} C_VEL
LIN {X 0,Y 578.53,Z 1204.214,A -85,B 0,C 180,E1 26750.201,E2 26750.201} C_VEL
LIN {X 0,Y 577.411,Z 1216.745,A -85,B 0,C 180,E1 26747.415,E2 26747.415} C_VEL
LIN {X 0,Y 576.8,Z 1225.666,A -85,B 0,C 180,E1 26745.066,E2 26745.066} C_VEL
LIN {X 0,Y 576.386,Z 1232.931,A -85,B 0,C 180,E1 26742.824,E2 26742.824} C_VEL
LIN {X 0,Y 576.141,Z 1238.972,A -85,B 0,C 180,E1 26740.595,E2 26740.595} C_VEL
LIN {X 0,Y 575.965,Z 1244.659,A -85,B 0,C 180,E1 26737.978,E2 26737.978} C_VEL
LIN {X 0,Y 575.925,Z 1248.608,A -85,B 0,C 180,E1 26735.375,E2 26735.375} C_VEL
LIN {X 0,Y 575.91,Z 1250.783,A -85,B 0,C 180,E1 26733.081,E2 26733.081} C_VEL
LIN {X 0,Y 575.885,Z 1251.75,A -85,B 0,C 180,E1 26731.09,E2 26731.09} C_VEL
LIN {X 0,Y 575.867,Z 1251.813,A -85,B 0,C 180,E1 26729.1,E2 26729.1} C_VEL
LIN {X 0,Y 575.909,Z 1250.975,A -85,B 0,C 180,E1 26727.11,E2 26727.11} C_VEL
LIN {X 0,Y 575.921,Z 1249.042,A -85,B 0,C 180,E1 26724.916,E2 26724.916} C_VEL
LIN {X 0,Y 575.955,Z 1245.647,A -85,B 0,C 180,E1 26722.514,E2 26722.514} C_VEL
LIN {X 0,Y 576.084,Z 1240.446,A -85,B 0,C 180,E1 26719.9,E2 26719.9} C_VEL
LIN {X 0,Y 576.34,Z 1233.778,A -85,B 0,C 180,E1 26717.369,E2 26717.369} C_VEL
LIN {X 0,Y 576.734,Z 1226.651,A -85,B 0,C 180,E1 26715.128,E2 26715.128} C_VEL
LIN {X 0,Y 577.259,Z 1218.626,A -85,B 0,C 180,E1 26712.968,E2 26712.968} C_VEL
LIN {X 0,Y 578.122,Z 1208.477,A -85,B 0,C 180,E1 26710.602,E2 26710.602} C_VEL
LIN {X 0,Y 579.456,Z 1194.937,A -85,B 0,C 180,E1 26707.9,E2 26707.9} C_VEL
LIN {X 0,Y 580.882,Z 1182.336,A -85,B 0,C 180,E1 26705.704,E2 26705.704} C_VEL
LIN {X 0,Y 582.718,Z 1168.137,A -85,B 0,C 180,E1 26703.501,E2 26703.501} C_VEL
LIN {X 0,Y 585.18,Z 1149.981,A -85,B 0,C 180,E1 26701.028,E2 26701.028} C_VEL
LIN {X 0,Y 587.491,Z 1134.168,A -85,B 0,C 180,E1 26699.123,E2 26699.123} C_VEL
LIN {X 0,Y 589.891,Z 1118.125,A -85,B 0,C 180,E1 26697.38,E2 26697.38} C_VEL
LIN {X 0,Y 592.993,Z 1098.112,A -85,B 0,C 180,E1 26695.428,E2 26695.428} C_VEL
LIN {X 0,Y 596.24,Z 1076.352,A -85,B 0,C 180,E1 26693.58,E2 26693.58} C_VEL
LIN {X 0,Y 598.947,Z 1058.279,A -85,B 0,C 180,E1 26692.214,E2 26692.214} C_VEL
LIN {X 0,Y 601.643,Z 1039.722,A -85,B 0,C 180,E1 26690.956,E2 26690.956} C_VEL
LIN {X 0,Y 604.685,Z 1018.016,A -85,B 0,C 180,E1 26689.653,E2 26689.653} C_VEL
LIN {X 0,Y 608.082,Z 991.792,A -85,B 0,C 180,E1 26688.305,E2 26688.305} C_VEL
LIN {X 0,Y 610.55,Z 970.644,A -85,B 0,C 180,E1 26687.373,E2 26687.373} C_VEL
LIN {X 0,Y 612.717,Z 950.21,A -85,B 0,C 180,E1 26686.602,E2 26686.602} C_VEL
LIN {X 0,Y 614.686,Z 929.032,A -85,B 0,C 180,E1 26685.926,E2 26685.926} C_VEL
LIN {X 0,Y 616.742,Z 903.3,A -85,B 0,C 180,E1 26685.261,E2 26685.261} C_VEL
LIN {X 0,Y 618.281,Z 876.019,A -85,B 0,C 180,E1 26684.748,E2 26684.748} C_VEL
LIN {X 0,Y 620.663,Z 793.216,A -85,B 0,C 180,E1 26683.582,E2 26683.582} C_VEL
LIN {X 0,Y 626.647,Z 577.396,A -85,B 0,C 180,E1 26680.548,E2 26680.548} C_VEL
LIN {X 0,Y 629.578,Z 477.561,A -85,B 0,C 180,E1 26679.118,E2 26679.118} C_VEL
LIN {X 0,Y 615.61,Z 458.347,A -85,B 0,C 180,E1 26677.114,E2 26677.114} C_VEL
LIN {X 0,Y 604.15,Z 443.42,A -85,B 0,C 180,E1 26675.341,E2 26675.341} C_VEL
LIN {X 0,Y 598.959,Z 437.009,A -85,B 0,C 180,E1 26674.495,E2 26674.495} C_VEL
LIN {X 0,Y 595.371,Z 432.434,A -85,B 0,C 180,E1 26673.888,E2 26673.888} C_VEL
LIN {X 0,Y 591.857,Z 427.801,A -85,B 0,C 180,E1 26673.274,E2 26673.274} C_VEL
LIN {X 0,Y 588.207,Z 423.85,A -85,B 0,C 180,E1 26672.636,E2 26672.636} C_VEL
LIN {X 0,Y 586.705,Z 421.592,A -85,B 0,C 180,E1 26672.353,E2 26672.353} C_VEL
LIN {X 0,Y 583.595,Z 418.504,A -85,B 0,C 180,E1 26671.793,E2 26671.793} C_VEL
LIN {X 0,Y 581.821,Z 415.536,A -85,B 0,C 180,E1 26671.439,E2 26671.439} C_VEL
LIN {X 0,Y 578.861,Z 413.105,A -85,B 0,C 180,E1 26670.894,E2 26670.894} C_VEL
LIN {X 0,Y 577.459,Z 410.143,A -85,B 0,C 180,E1 26670.588,E2 26670.588} C_VEL
LIN {X 0,Y 577.302,Z 409.275,A -85,B 0,C 180,E1 26670.519,E2 26670.519} C_VEL
LIN {X 0,Y 577.303,Z 409.307,A -85,B 0,C 180,E1 26667.309,E2 26667.309} C_VEL
LIN {X 0,Y 577.313,Z 409.295,A -85,B 0,C 180,E1 26664.018,E2 26664.018} C_VEL
LIN {X 0,Y 577.309,Z 409.272,A -85,B 0,C 180,E1 26660.691,E2 26660.691} C_VEL
LIN {X 0,Y 577.308,Z 409.319,A -85,B 0,C 180,E1 26657.332,E2 26657.332} C_VEL
LIN {X 0,Y 577.307,Z 409.274,A -85,B 0,C 180,E1 26654.033,E2 26654.033} C_VEL
LIN {X 0,Y 577.295,Z 409.304,A -85,B 0,C 180,E1 26650.781,E2 26650.781} C_VEL
LIN {X 0,Y 577.313,Z 409.285,A -85,B 0,C 180,E1 26647.464,E2 26647.464} C_VEL
LIN {X 0,Y 577.301,Z 409.285,A -85,B 0,C 180,E1 26644.172,E2 26644.172} C_VEL
LIN {X 0,Y 577.303,Z 409.305,A -85,B 0,C 180,E1 26640.794,E2 26640.794} C_VEL
LIN {X 0,Y 577.309,Z 409.27,A -85,B 0,C 180,E1 26637.518,E2 26637.518} C_VEL
LIN {X 0,Y 577.29,Z 409.314,A -85,B 0,C 180,E1 26634.234,E2 26634.234} C_VEL
LIN {X 0,Y 577.309,Z 409.266,A -85,B 0,C 180,E1 26631.032,E2 26631.032} C_VEL
LIN {X 0,Y 577.291,Z 409.32,A -85,B 0,C 180,E1 26627.801,E2 26627.801} C_VEL
LIN {X 0,Y 577.315,Z 409.272,A -85,B 0,C 180,E1 26624.531,E2 26624.531} C_VEL
LIN {X 0,Y 577.301,Z 409.299,A -85,B 0,C 180,E1 26621.311,E2 26621.311} C_VEL
LIN {X 0,Y 577.29,Z 409.308,A -85,B 0,C 180,E1 26617.921,E2 26617.921} C_VEL
LIN {X 0,Y 577.314,Z 409.273,A -85,B 0,C 180,E1 26614.672,E2 26614.672} C_VEL
LIN {X 0,Y 577.281,Z 409.294,A -85,B 0,C 180,E1 26611.424,E2 26611.424} C_VEL
LIN {X 0,Y 577.284,Z 409.3,A -85,B 0,C 180,E1 26611.159,E2 26611.159} C_VEL
LIN {X 0,Y 578.64,Z 412.782,A -85,B 0,C 180,E1 26610.496,E2 26610.496} C_VEL
LIN {X 0,Y 580.057,Z 414.875,A -85,B 0,C 180,E1 26610.007,E2 26610.007} C_VEL
LIN {X 0,Y 581.794,Z 418.387,A -85,B 0,C 180,E1 26609.307,E2 26609.307} C_VEL
LIN {X 0,Y 582.858,Z 420.332,A -85,B 0,C 180,E1 26608.911,E2 26608.911} C_VEL
LIN {X 0,Y 584.596,Z 423.345,A -85,B 0,C 180,E1 26608.354,E2 26608.354} C_VEL
LIN {X 0,Y 589.191,Z 429.22,A -85,B 0,C 180,E1 26607.512,E2 26607.512} C_VEL
LIN {X 0,Y 602.07,Z 446.609,A -85,B 0,C 180,E1 26605.293,E2 26605.293} C_VEL
LIN {X 0,Y 612.525,Z 461.314,A -85,B 0,C 180,E1 26603.632,E2 26603.632} C_VEL
LIN {X 0,Y 623.138,Z 476.92,A -85,B 0,C 180,E1 26602.05,E2 26602.05} C_VEL
LIN {X 0,Y 629.82,Z 487.382,A -85,B 0,C 180,E1 26601.098,E2 26601.098} C_VEL
LIN {X 0,Y 623.757,Z 701.096,A -85,B 0,C 180,E1 26598.061,E2 26598.061} C_VEL
LIN {X 0,Y 618.263,Z 903.017,A -85,B 0,C 180,E1 26595.24,E2 26595.24} C_VEL
LIN {X 0,Y 616.965,Z 926.806,A -85,B 0,C 180,E1 26594.812,E2 26594.812} C_VEL
LIN {X 0,Y 614.806,Z 955.63,A -85,B 0,C 180,E1 26594.108,E2 26594.108} C_VEL
LIN {X 0,Y 612.812,Z 977.649,A -85,B 0,C 180,E1 26593.422,E2 26593.422} C_VEL
LIN {X 0,Y 610.721,Z 997.946,A -85,B 0,C 180,E1 26592.676,E2 26592.676} C_VEL
LIN {X 0,Y 608.558,Z 1017.39,A -85,B 0,C 180,E1 26591.845,E2 26591.845} C_VEL
LIN {X 0,Y 606.27,Z 1035.977,A -85,B 0,C 180,E1 26590.943,E2 26590.943} C_VEL
LIN {X 0,Y 603.668,Z 1055.467,A -85,B 0,C 180,E1 26589.87,E2 26589.87} C_VEL
LIN {X 0,Y 600.526,Z 1078.053,A -85,B 0,C 180,E1 26588.457,E2 26588.457} C_VEL
LIN {X 0,Y 597.058,Z 1101.175,A -85,B 0,C 180,E1 26586.78,E2 26586.78} C_VEL
LIN {X 0,Y 594.21,Z 1119.786,A -85,B 0,C 180,E1 26585.255,E2 26585.255} C_VEL
LIN {X 0,Y 591.558,Z 1137.12,A -85,B 0,C 180,E1 26583.673,E2 26583.673} C_VEL
LIN {X 0,Y 588.541,Z 1157.308,A -85,B 0,C 180,E1 26581.612,E2 26581.612} C_VEL
LIN {X 0,Y 585.844,Z 1175.471,A -85,B 0,C 180,E1 26579.489,E2 26579.489} C_VEL
LIN {X 0,Y 583.724,Z 1190.353,A -85,B 0,C 180,E1 26577.552,E2 26577.552} C_VEL
LIN {X 0,Y 581.685,Z 1206.257,A -85,B 0,C 180,E1 26575.236,E2 26575.236} C_VEL
LIN {X 0,Y 579.858,Z 1221.395,A -85,B 0,C 180,E1 26572.699,E2 26572.699} C_VEL
LIN {X 0,Y 578.648,Z 1232.865,A -85,B 0,C 180,E1 26570.517,E2 26570.517} C_VEL
LIN {X 0,Y 577.68,Z 1243.345,A -85,B 0,C 180,E1 26568.261,E2 26568.261} C_VEL
LIN {X 0,Y 576.872,Z 1254.38,A -85,B 0,C 180,E1 26565.481,E2 26565.481} C_VEL
LIN {X 0,Y 576.433,Z 1262.129,A -85,B 0,C 180,E1 26563.138,E2 26563.138} C_VEL
LIN {X 0,Y 576.157,Z 1268.045,A -85,B 0,C 180,E1 26561.009,E2 26561.009} C_VEL
LIN {X 0,Y 576.011,Z 1273.121,A -85,B 0,C 180,E1 26558.791,E2 26558.791} C_VEL
LIN {X 0,Y 575.945,Z 1277.628,A -85,B 0,C 180,E1 26556.183,E2 26556.183} C_VEL
LIN {X 0,Y 575.913,Z 1280.468,A -85,B 0,C 180,E1 26553.588,E2 26553.588} C_VEL
LIN {X 0,Y 575.895,Z 1281.713,A -85,B 0,C 180,E1 26551.298,E2 26551.298} C_VEL
LIN {X 0,Y 575.864,Z 1281.828,A -85,B 0,C 180,E1 26549.209,E2 26549.209} C_VEL
LIN {X 0,Y 575.91,Z 1281.018,A -85,B 0,C 180,E1 26547.218,E2 26547.218} C_VEL
LIN {X 0,Y 575.921,Z 1279.114,A -85,B 0,C 180,E1 26545.025,E2 26545.025} C_VEL
LIN {X 0,Y 575.962,Z 1275.909,A -85,B 0,C 180,E1 26542.724,E2 26542.724} C_VEL
LIN {X 0,Y 576.06,Z 1270.828,A -85,B 0,C 180,E1 26540.11,E2 26540.11} C_VEL
LIN {X 0,Y 576.325,Z 1263.974,A -85,B 0,C 180,E1 26537.48,E2 26537.48} C_VEL
LIN {X 0,Y 576.714,Z 1256.88,A -85,B 0,C 180,E1 26535.24,E2 26535.24} C_VEL
LIN {X 0,Y 577.235,Z 1248.918,A -85,B 0,C 180,E1 26533.087,E2 26533.087} C_VEL
LIN {X 0,Y 578.04,Z 1239.248,A -85,B 0,C 180,E1 26530.817,E2 26530.817} C_VEL
LIN {X 0,Y 579.355,Z 1225.899,A -85,B 0,C 180,E1 26528.119,E2 26528.119} C_VEL
LIN {X 0,Y 580.813,Z 1212.901,A -85,B 0,C 180,E1 26525.842,E2 26525.842} C_VEL
LIN {X 0,Y 582.451,Z 1200.017,A -85,B 0,C 180,E1 26523.827,E2 26523.827} C_VEL
LIN {X 0,Y 584.729,Z 1183.457,A -85,B 0,C 180,E1 26521.511,E2 26521.511} C_VEL
LIN {X 0,Y 587.332,Z 1165.204,A -85,B 0,C 180,E1 26519.286,E2 26519.286} C_VEL
LIN {X 0,Y 589.713,Z 1149.281,A -85,B 0,C 180,E1 26517.545,E2 26517.545} C_VEL
LIN {X 0,Y 592.328,Z 1132.226,A -85,B 0,C 180,E1 26515.863,E2 26515.863} C_VEL
LIN {X 0,Y 595.725,Z 1109.969,A -85,B 0,C 180,E1 26513.912,E2 26513.912} C_VEL
LIN {X 0,Y 598.81,Z 1089.19,A -85,B 0,C 180,E1 26512.325,E2 26512.325} C_VEL
LIN {X 0,Y 601.589,Z 1070.079,A -85,B 0,C 180,E1 26511.025,E2 26511.025} C_VEL
LIN {X 0,Y 604.495,Z 1049.331,A -85,B 0,C 180,E1 26509.774,E2 26509.774} C_VEL
LIN {X 0,Y 607.849,Z 1023.411,A -85,B 0,C 180,E1 26508.429,E2 26508.429} C_VEL
LIN {X 0,Y 610.416,Z 1000.769,A -85,B 0,C 180,E1 26507.437,E2 26507.437} C_VEL
LIN {X 0,Y 612.556,Z 980.173,A -85,B 0,C 180,E1 26506.664,E2 26506.664} C_VEL
